(* IEC 61131-3 sources: MotionTestBenchMaster/Logical/00_AID/Libraries/Sidel_Libraries/Sidel_Obj (part 2) *)

(* ---- Shift_Obj.st ---- *)
FUNCTION_BLOCK PhotoCell_SftObj
	IF IN_ConfigPresent THEN
		VAR_GrippersNumber	:= LIMIT(1, IN_GrippersNumber, CST_RepetitiveArrayDim);
		VAR_Mask 			:= IN_MaskEn AND HMI.Mask;

		IF VAR_Mask THEN
			VAR_Signal := IN_WaitOn AND NOT IN_WaitOff;
		ELSE
			VAR_Signal := IO.DI_Input;
		END_IF

		HMI.On := VAR_Signal;

		OUT	:= HMI.On;

		IF IN_MachinePitch AND IN_Enable THEN
			VAR_ActualValveCounter	:= INT_TO_USINT(FC_ReminderShift(VAR_ActualValveCounter	+ 1, VAR_GrippersNumber, 0));

			IF IN_WritePresenceEnable THEN //v1.63
				SHIFT_Position.ContainerPresence	:= IO.DI_Input;
			END_IF//v1.63

			IF SHIFT_Position.ContainerPresence THEN//v1.63
				IF NOT SHIFT_Position.ContainerBurst	AND	NOT VAR_Mask THEN//v1.63
					IF NOT IO.DI_Input THEN
						HMI.ConsecutiveErrors	:= SEL((IN_MStopConsecutiveValue > 0), 0,HMI.ConsecutiveErrors + 1);
						HMI.AbsoluteErrors		:= SEL((IN_CBlockAbsoluteValue > 0), 0, HMI.AbsoluteErrors + 1);
						HMI.TotalErrors			:= SEL((IN_MStopAbsoluteValue > 0), HMI.TotalErrors, HMI.TotalErrors + 1);

						VAR_RepetitiveCounterArray[VAR_ActualValveCounter]	:= SEL((IN_CBlockRepetitiveValue > 0), 0, VAR_RepetitiveCounterArray[VAR_ActualValveCounter] + 1);
						SHIFT_Position.ContainerPresence	:= FALSE;//v1.63

						IF VAR_RepetitiveCounterArray[VAR_ActualValveCounter] > IN_CBlockRepetitiveValue THEN
							OUT_CBlockRepetitive	:= TRUE;
						END_IF
					ELSE
						VAR_RepetitiveCounterArray[VAR_ActualValveCounter]	:= 0;
						HMI.ConsecutiveErrors	:= 0;//v1.63
					END_IF
				ELSE//v1.63
					VAR_RepetitiveCounterArray[VAR_ActualValveCounter]	:= 0;
					HMI.ConsecutiveErrors	:= 0;
				END_IF//v1.63
			END_IF

			HMI.AlwaysTrueSteps	:= SEL(VAR_EdgeChecked, HMI.AlwaysTrueSteps + 1, 0);//v1.63

			IF IN_CBlockRepetitiveValue > 0 THEN
				HMI.RepetitiveErrors	:= 0;

				FOR VAR_GrippersNumber:= 1	TO	CST_RepetitiveArrayDim	DO
					HMI.RepetitiveErrors := MAX(HMI.RepetitiveErrors, VAR_RepetitiveCounterArray[VAR_GrippersNumber]);
				END_FOR
			END_IF
		ELSIF NOT IO.DI_Input AND IN_Enable THEN
			VAR_EdgeChecked		:= TRUE;
		END_IF

		TMR_TON_TotalCounterReset(IN := IN_ResetCounters OR HMI.CounterReset, PT := T#5s);

		IF IN_ResetCounters OR HMI.CounterReset OR VAR_Mask OR NOT IN_Enable THEN
			IF NOT VAR_CounterResetMemory THEN
				VAR_CounterResetMemory	:= TRUE;

				FOR VAR_GrippersNumber:= 1 TO CST_RepetitiveArrayDim DO
					VAR_RepetitiveCounterArray[VAR_GrippersNumber]	:= 0;
					OUT_CBlockRepetitive	:= FALSE;
				END_FOR

				HMI.AlwaysTrueSteps		:= 0;
				HMI.RepetitiveErrors	:= 0;
				HMI.ConsecutiveErrors	:= 0;
				HMI.AbsoluteErrors		:= 0;
			END_IF
		ELSE
			VAR_CounterResetMemory	:= FALSE;
		END_IF

		IF TMR_TON_TotalCounterReset.Q THEN
			IF NOT VAR_TotalCounterResetMemory THEN
				VAR_TotalCounterResetMemory := TRUE;
				HMI.TotalErrors	:= 0;
			END_IF
		ELSE
			VAR_TotalCounterResetMemory := FALSE;
		END_IF

		HMI.ConfigPresent 	:= IN_ConfigPresent;
		HMI.ConfigAlarm 	:= IN_Alarm;
		HMI.Alarm 			:= OUT_CBlockAbsolute OR OUT_MStopConsecutive OR OUT_MStopAbsolute OR OUT_AlwaysTrueError;
		HMI.Wait			:= (IN_WaitOn AND NOT HMI.On) OR (IN_WaitOff AND HMI.On);
		HMI.MaskEnable		:= IN_MaskEn;

		OUT_CBlockAbsolute		:= (HMI.AbsoluteErrors 		>= IN_CBlockAbsoluteValue)		AND (IN_CBlockAbsoluteValue		> 0);
		OUT_MStopConsecutive	:= (HMI.ConsecutiveErrors 	>= IN_MStopConsecutiveValue)	AND (IN_MStopConsecutiveValue	> 0);
		OUT_MStopAbsolute		:= (HMI.AbsoluteErrors 		>= (IN_MStopAbsoluteValue + IN_CBlockAbsoluteValue))		AND (IN_MStopAbsoluteValue		> 0);	//V4.A.A.1.6.12
		OUT_AlwaysTrueError		:= (HMI.AlwaysTrueSteps		>= CST_AlwaysTrueMaxSteps)		AND (CST_AlwaysTrueMaxSteps		> 0);
	ELSE
		OUT						:= FALSE;
		OUT_CBlockRepetitive	:= FALSE;
		OUT_CBlockAbsolute		:= FALSE;
		OUT_MStopConsecutive	:= FALSE;
		OUT_MStopAbsolute		:= FALSE;
		OUT_AlwaysTrueError		:= FALSE;
		HMI.On 					:= FALSE;
		HMI.MaskEnable			:= FALSE;
		HMI.ConfigPresent 		:= FALSE;
		HMI.ConfigAlarm 		:= FALSE;
		HMI.Alarm 				:= FALSE;
		HMI.Wait				:= FALSE;
		HMI.RepetitiveErrors	:= 0;
		HMI.ConsecutiveErrors	:= 0;
		HMI.AbsoluteErrors		:= 0;
		HMI.AlwaysTrueSteps		:= 0;
	END_IF
END_FUNCTION_BLOCK

FUNCTION_BLOCK CapPhotoCell_SftObj
	IF IN_ConfigPresent THEN
		VAR_GrippersNumber	:= LIMIT(1, IN_GrippersNumber, CST_CounterArrayDim);
		VAR_Mask 			:= IN_MaskEn AND HMI.Mask;

		IF VAR_Mask THEN
			VAR_Signal := IN_WaitOn AND NOT IN_WaitOff;
		ELSE
			VAR_Signal := IO.DI_Input;
		END_IF

		HMI.On := VAR_Signal;

		OUT	:= HMI.On;

		IF IN_MachinePitch AND IN_Enable THEN
			VAR_ActualValveCounter	:= INT_TO_USINT(FC_ReminderShift(VAR_ActualValveCounter + 1, VAR_GrippersNumber, 0));

			IF SHIFT_Position.ContainerPresence AND SHIFT_Position.ClosingReleased AND NOT VAR_Mask THEN
				HMI.AlwaysTrueSteps	:= SEL(VAR_EdgeChecked, HMI.AlwaysTrueSteps + 1, 0);
				SHIFT_Position.ContainerClosed	:= IO.DI_Input;

				IF VAR_CapsReleased < 16#FFFFFFFF THEN
					VAR_CapsReleased := VAR_CapsReleased + 1;
				ELSE
					FOR VAR_i := VAR_AbsoluteErrorN TO 1 BY -1 DO
						VAR_AbsoluteCounterArray[VAR_i] := VAR_AbsoluteCounterArray[VAR_i] - (VAR_AbsoluteCounterArray[1] - 1);
					END_FOR
					VAR_CapsReleased := VAR_AbsoluteCounterArray[VAR_AbsoluteErrorN] + 1;
				END_IF

				IF NOT IO.DI_Input THEN
					HMI.ConsecutiveErrors	:= SEL((IN_MStopConsecutiveValue > 0), 0,HMI.ConsecutiveErrors + 1);
					//HMI.AbsoluteErrors		:= SEL((IN_CBlockAbsoluteValue > 0), 0, VAR_AbsoluteErrorN);	//V4.A.A.1.6.12
					HMI.TotalErrors			:= SEL((IN_CBlockAbsoluteValue > 0) OR (IN_MStopConsecutiveValue > 0), HMI.TotalErrors, HMI.TotalErrors + 1);

					VAR_RepetitiveCounterArray[VAR_ActualValveCounter] := SEL((IN_CBlockRepetitiveValue > 0), 0, VAR_RepetitiveCounterArray[VAR_ActualValveCounter] + 1);

					IF VAR_RepetitiveCounterArray[VAR_ActualValveCounter] > IN_CBlockRepetitiveValue THEN
						OUT_CBlockRepetitive	:= TRUE;
					END_IF

					IF IN_CBlockAbsoluteValue > 0 THEN
						IF IN_CBlockAbsoluteQuantity > 0 THEN
							VAR_AbsoluteCounterArray[VAR_AbsoluteErrorN] := VAR_CapsReleased;
						ELSE
							VAR_AbsoluteCounterArray[VAR_AbsoluteErrorN] := 0;
						END_IF

						VAR_AbsoluteErrorN := VAR_AbsoluteErrorN + 1;
					ELSE
						VAR_AbsoluteCounterArray[VAR_AbsoluteErrorN] := 0;
						VAR_AbsoluteErrorN := 1;
					END_IF
				ELSE
					VAR_RepetitiveCounterArray[VAR_ActualValveCounter]	:= 0;
				END_IF
			ELSE
				HMI.ConsecutiveErrors	:= 0;
			END_IF

			IF ((VAR_CapsReleased - VAR_AbsoluteCounterArray[1]) > IN_CBlockAbsoluteQuantity) AND (IN_CBlockAbsoluteQuantity > 0) THEN
				memmove(ADR(VAR_AbsoluteCounterArray[1]), ADR(VAR_AbsoluteCounterArray[2]), SIZEOF(VAR_AbsoluteCounterArray[1]) * 49);
				VAR_AbsoluteCounterArray[50] := 0;
				VAR_AbsoluteErrorN := MAX(VAR_AbsoluteErrorN - 1, 1);
			END_IF

			IF IN_CBlockRepetitiveValue > 0 THEN
				HMI.RepetitiveErrors := 0;
				FOR VAR_GrippersNumber:= 1 TO CST_CounterArrayDim DO
					HMI.RepetitiveErrors := MAX(HMI.RepetitiveErrors, VAR_RepetitiveCounterArray[VAR_GrippersNumber]);
				END_FOR
			END_IF

			HMI.AbsoluteErrors		:= SEL((IN_CBlockAbsoluteValue > 0), 0, VAR_AbsoluteErrorN - 1);	//V4.A.A.1.6.12
		ELSIF NOT IO.DI_Input AND IN_Enable THEN
			VAR_EdgeChecked := TRUE;
		ELSIF NOT IN_Enable THEN
			SHIFT_Position.ContainerClosed	:= SHIFT_Position.ContainerPresence AND SHIFT_Position.ClosingReleased;
		END_IF

		TMR_TON_TotalCounterReset(IN := IN_ResetCounters OR HMI.CounterReset, PT := T#5s);

		IF IN_ResetCounters OR HMI.CounterReset OR VAR_Mask OR NOT IN_Enable THEN
			IF NOT VAR_CounterResetMemory THEN
				VAR_CounterResetMemory	:= TRUE;

				FOR VAR_GrippersNumber:= 1 TO CST_CounterArrayDim DO
					VAR_RepetitiveCounterArray[VAR_GrippersNumber]	:= 0;
					OUT_CBlockRepetitive	:= FALSE;
				END_FOR

				memset(ADR(VAR_AbsoluteCounterArray[1]), 0, SIZEOF(VAR_AbsoluteCounterArray));
				VAR_AbsoluteErrorN := 1;

				VAR_CapsReleased		:= 0;
				HMI.AlwaysTrueSteps		:= 0;
				HMI.RepetitiveErrors	:= 0;
				//HMI.ConsecutiveErrors	:= 0;//V1.61
				HMI.AbsoluteErrors		:= 0;
			END_IF
		ELSE
			VAR_CounterResetMemory	:= FALSE;
		END_IF
		(*V1.61 Consecutive Errorors counter reset new management*)
		IF IN_ResetCountersConsecutive OR VAR_Mask OR NOT IN_Enable THEN
			IF NOT VAR_CounterConsResetMemory THEN
				VAR_CounterConsResetMemory	:= TRUE;
				HMI.ConsecutiveErrors	:= 0;
			END_IF
		ELSE
			VAR_CounterConsResetMemory	:= FALSE;
		END_IF

		IF TMR_TON_TotalCounterReset.Q THEN
			IF NOT VAR_TotalCounterResetMemory THEN
				VAR_TotalCounterResetMemory := TRUE;
				HMI.TotalErrors	:= 0;
			END_IF
		ELSE
			VAR_TotalCounterResetMemory := FALSE;
		END_IF

		HMI.ConfigPresent 	:= IN_ConfigPresent;
		HMI.ConfigAlarm 	:= IN_Alarm;
		HMI.Alarm 			:= OUT_CBlockAbsolute OR OUT_MStopConsecutive OR OUT_AlwaysTrueError;
		HMI.Wait			:= (IN_WaitOn AND NOT HMI.On) OR (IN_WaitOff AND HMI.On);
		HMI.MaskEnable		:= IN_MaskEn;

		OUT_CBlockAbsolute		:= (HMI.AbsoluteErrors 		>= IN_CBlockAbsoluteValue)		AND (IN_CBlockAbsoluteValue		> 0);
		OUT_MStopConsecutive	:= (HMI.ConsecutiveErrors 	>= IN_MStopConsecutiveValue)	AND (IN_MStopConsecutiveValue	> 0);
		OUT_AlwaysTrueError		:= (HMI.AlwaysTrueSteps		>= CST_AlwaysTrueMaxSteps)		AND (CST_AlwaysTrueMaxSteps		> 0);
	ELSE
		OUT						:= FALSE;
		OUT_CBlockRepetitive	:= FALSE;
		OUT_CBlockAbsolute		:= FALSE;
		OUT_MStopConsecutive	:= FALSE;
		OUT_AlwaysTrueError		:= FALSE;
		HMI.On 					:= FALSE;
		HMI.MaskEnable			:= FALSE;
		HMI.ConfigPresent 		:= FALSE;
		HMI.ConfigAlarm 		:= FALSE;
		HMI.Alarm 				:= FALSE;
		HMI.Wait				:= FALSE;
		HMI.RepetitiveErrors	:= 0;
		HMI.ConsecutiveErrors	:= 0;
		HMI.AbsoluteErrors		:= 0;
		HMI.AlwaysTrueSteps		:= 0;
	END_IF
END_FUNCTION_BLOCK

FUNCTION_BLOCK CapPhotoCell_SftObj_old
	IF IN_ConfigPresent THEN
		VAR_GrippersNumber	:= LIMIT(1, IN_GrippersNumber, CST_RepetitiveArrayDim);
		VAR_Mask 			:= IN_MaskEn AND HMI.Mask;

		IF VAR_Mask THEN
			VAR_Signal := IN_WaitOn AND NOT IN_WaitOff;
		ELSE
			VAR_Signal := IO.DI_Input;
		END_IF

		HMI.On := VAR_Signal;

		OUT	:= HMI.On;

		IF IN_MachinePitch AND IN_Enable THEN
			VAR_ActualValveCounter	:= INT_TO_USINT(FC_ReminderShift(VAR_ActualValveCounter + 1, VAR_GrippersNumber, 0));

			IF SHIFT_Position.ContainerPresence AND SHIFT_Position.ClosingReleased AND NOT VAR_Mask THEN
				HMI.AlwaysTrueSteps	:= SEL(VAR_EdgeChecked, HMI.AlwaysTrueSteps + 1, 0);
				SHIFT_Position.ContainerClosed	:= IO.DI_Input;

				IF NOT IO.DI_Input THEN
					HMI.ConsecutiveErrors	:= SEL((IN_MStopConsecutiveValue > 0), 0,HMI.ConsecutiveErrors + 1);
					HMI.AbsoluteErrors		:= SEL((IN_CBlockAbsoluteValue > 0), 0, HMI.AbsoluteErrors + 1);
					HMI.TotalErrors			:= SEL((IN_MStopAbsoluteValue > 0), HMI.TotalErrors, HMI.TotalErrors + 1);

					VAR_RepetitiveCounterArray[VAR_ActualValveCounter] := SEL((IN_CBlockRepetitiveValue > 0), 0, VAR_RepetitiveCounterArray[VAR_ActualValveCounter] + 1);

					IF VAR_RepetitiveCounterArray[VAR_ActualValveCounter] > IN_CBlockRepetitiveValue THEN
						OUT_CBlockRepetitive	:= TRUE;
					END_IF
				ELSE
					VAR_RepetitiveCounterArray[VAR_ActualValveCounter]	:= 0;
				END_IF
			ELSE
				HMI.ConsecutiveErrors	:= 0;
			END_IF

			IF IN_CBlockRepetitiveValue > 0 THEN
				HMI.RepetitiveErrors := 0;
				FOR VAR_GrippersNumber:= 1 TO CST_RepetitiveArrayDim DO
					HMI.RepetitiveErrors := MAX(HMI.RepetitiveErrors, VAR_RepetitiveCounterArray[VAR_GrippersNumber]);
				END_FOR
			END_IF
		ELSIF NOT IO.DI_Input AND IN_Enable THEN
			VAR_EdgeChecked := TRUE;
		ELSIF NOT IN_Enable THEN
			SHIFT_Position.ContainerClosed	:= SHIFT_Position.ContainerPresence AND SHIFT_Position.ClosingReleased;
		END_IF

		TMR_TON_TotalCounterReset(IN := IN_ResetCounters OR HMI.CounterReset, PT := T#5s);

		IF IN_ResetCounters OR HMI.CounterReset OR VAR_Mask THEN
			IF NOT VAR_CounterResetMemory THEN
				VAR_CounterResetMemory	:= TRUE;

				FOR VAR_GrippersNumber:= 1 TO CST_RepetitiveArrayDim DO
					VAR_RepetitiveCounterArray[VAR_GrippersNumber]	:= 0;
					OUT_CBlockRepetitive	:= FALSE;
				END_FOR

				HMI.AlwaysTrueSteps		:= 0;
				HMI.RepetitiveErrors	:= 0;
				HMI.ConsecutiveErrors	:= 0;
				HMI.AbsoluteErrors		:= 0;
			END_IF
		ELSE
			VAR_CounterResetMemory	:= FALSE;
		END_IF

		IF TMR_TON_TotalCounterReset.Q THEN
			IF NOT VAR_TotalCounterResetMemory THEN
				VAR_TotalCounterResetMemory := TRUE;
				HMI.TotalErrors	:= 0;
			END_IF
		ELSE
			VAR_TotalCounterResetMemory := FALSE;
		END_IF

		HMI.ConfigPresent 	:= IN_ConfigPresent;
		HMI.ConfigAlarm 	:= IN_Alarm;
		HMI.Alarm 			:= OUT_CBlockAbsolute OR OUT_MStopConsecutive OR OUT_MStopAbsolute OR OUT_AlwaysTrueError;
		HMI.Wait			:= (IN_WaitOn AND NOT HMI.On) OR (IN_WaitOff AND HMI.On);
		HMI.MaskEnable		:= IN_MaskEn;

		OUT_CBlockAbsolute		:= (HMI.AbsoluteErrors 		>= IN_CBlockAbsoluteValue)		AND (IN_CBlockAbsoluteValue		> 0);
		OUT_MStopConsecutive	:= (HMI.ConsecutiveErrors 	>= IN_MStopConsecutiveValue)	AND (IN_MStopConsecutiveValue	> 0);
		OUT_MStopAbsolute		:= (HMI.AbsoluteErrors 		>= IN_MStopAbsoluteValue)		AND (IN_MStopAbsoluteValue		> 0);
		OUT_AlwaysTrueError		:= (HMI.AlwaysTrueSteps		>= CST_AlwaysTrueMaxSteps)		AND (CST_AlwaysTrueMaxSteps		> 0);
	ELSE
		OUT						:= FALSE;
		OUT_CBlockRepetitive	:= FALSE;
		OUT_CBlockAbsolute		:= FALSE;
		OUT_MStopConsecutive	:= FALSE;
		OUT_MStopAbsolute		:= FALSE;
		OUT_AlwaysTrueError		:= FALSE;
		HMI.On 					:= FALSE;
		HMI.MaskEnable			:= FALSE;
		HMI.ConfigPresent 		:= FALSE;
		HMI.ConfigAlarm 		:= FALSE;
		HMI.Alarm 				:= FALSE;
		HMI.Wait				:= FALSE;
		HMI.RepetitiveErrors	:= 0;
		HMI.ConsecutiveErrors	:= 0;
		HMI.AbsoluteErrors		:= 0;
		HMI.AlwaysTrueSteps		:= 0;
	END_IF
END_FUNCTION_BLOCK

FUNCTION_BLOCK Ejector_SftObj
	VAR_Mask	:= HMI.Mask AND IN_MaskEn;

	(* Local *)
	IF IN_ManEn AND NOT IN_HMIAutoForce THEN
		VAR_ManOn	:= HMI.ManOn;
		VAR_Auto	:= NOT HMI.ManOff AND NOT HMI.ManOn;
	ELSE
		VAR_ManOn	:= FALSE;
		VAR_Auto	:= TRUE;
		HMI.ManOn	:= FALSE;
		HMI.ManOff	:= FALSE;
	END_IF

	IF IN_MachinePitch THEN
		VAR_AutoCnd := IN_ShiftPosition.ContainerPresence		AND (IN_ShiftPosition.ContainerBurst	OR
						(NOT IN_ShiftPosition.ContainerFilled	AND IN_FillingErrorEject) OR IN_ShiftPosition.EjectContainer) AND NOT VAR_Mask; (*V1.61*)
		IF VAR_AutoCnd AND NOT IN_SamplingModeActive THEN (*V1.61*)
			HMI.ConsecutiveErrors	:= HMI.ConsecutiveErrors	+ 1;
			HMI.AbsoluteErrors		:= HMI.AbsoluteErrors		+ 1;
			HMI.TotalErrors			:= HMI.TotalErrors			+ 1;
		ELSE
			HMI.ConsecutiveErrors	:= 0;
		END_IF(*V1.61*)

		IF IN_SamplingModeActive AND VAR_AutoCnd THEN (*V1.61*)
			IN_ShiftPosition.ContainerEjected := TRUE;(*V1.61*)
		ELSE
			IN_ShiftPosition.ContainerEjected := FALSE;(*V1.61*)
		END_IF
	END_IF

	TMR_TON_TotalCounterReset(IN := IN_ResetCounters OR HMI.CounterReset, PT := T#5s);

	IF IN_ResetCounters OR HMI.CounterReset THEN
		IF NOT VAR_CounterResetMemory THEN
			VAR_CounterResetMemory	:= TRUE;
			HMI.ConsecutiveErrors	:= 0;
			HMI.AbsoluteErrors		:= 0;
		END_IF
	ELSE
		VAR_CounterResetMemory	:= FALSE;
	END_IF

	IF TMR_TON_TotalCounterReset.Q THEN
		IF NOT VAR_TotalCounterResetMemory THEN
			VAR_TotalCounterResetMemory := TRUE;
			HMI.TotalErrors	:= 0;
		END_IF
	ELSE
		VAR_TotalCounterResetMemory := FALSE;
	END_IF

	IF IN_ConfigPresent THEN
		IF IN_Enable THEN
			IF VAR_Auto THEN
				VAR_ValveOpened := VAR_AutoCnd;
			ELSIF VAR_ManOn THEN
				VAR_ValveOpened := TRUE;
			ELSE
				VAR_ValveOpened := FALSE;
			END_IF
		ELSIF NOT IN_ConfigType THEN
			VAR_ValveOpened := FALSE;
		END_IF
		VAR_ValveClosed := NOT VAR_ValveOpened;

		OUT						:= VAR_ValveOpened;
		OUT_CBlockAbsolute		:= (HMI.AbsoluteErrors 		>= IN_CBlockAbsoluteValue)		AND (IN_CBlockAbsoluteValue		> 0);
		OUT_MStopConsecutive	:= (HMI.ConsecutiveErrors 	>= IN_MStopConsecutiveValue)	AND (IN_MStopConsecutiveValue	> 0);
	ELSE
		VAR_ValveOpened			:= FALSE;
		VAR_ValveClosed			:= FALSE;
		OUT						:= FALSE;
		OUT_CBlockAbsolute		:= 0;
		OUT_MStopConsecutive	:= 0;
	END_IF

	(* HMI *)
	HMI.ManEnable		:= IN_ManEn;
	HMI.ConfigPresent	:= IN_ConfigPresent;
	HMI.MaskEnable		:= IN_MaskEn;
	HMI.Alarm 			:= OUT_CBlockAbsolute OR OUT_MStopConsecutive;

	(* IO *)
	IO.DO_Opened	:= VAR_ValveOpened;
	IO.DO_Closed	:= VAR_ValveClosed;
	HMI.Out			:= IO.DO_Opened;
END_FUNCTION_BLOCK

(* ---- Sidel_Obj.fun ---- *)
FUNCTION_BLOCK Analog_In_Direct_Inverse
	VAR_INPUT
		IN_ConfigPresent : BOOL;
		IN_Simulation : BOOL;
		IN_0_20mA : BOOL;
		IN_FaultOutMode : USINT; (*LowOnFault(1) ; HighOnFault (2) HoldOnFault (0)*)
		IN_EngScale : BOOL;
		IN_CompareMode : USINT; (*0 = Off, 1 = PV_Greater_SP, 2 = PV_Less_SP, 3 = PV_Equal_SP, 4 = On*)
		IN_ScaleLOW : REAL;
		IN_ScaleHIGH : REAL;
		IN_AlarmEn : BOOL;
		IN_MaskEn : BOOL;
		IN_ConfigPopup : BOOL;
		IN_Reset : BOOL; (*Reset Analog Channel Alarm*)
		IN_ActualSP : REAL; (*Signal Input Actual Set Point*)
		IN_MinDev : REAL; (*To Set Point Low Deviation (for SP obtained)*)
		IN_MaxDev : REAL; (*To Set Point High Deviation (for SP obtained)*)
		IN_WaitDelay : TIME;
		IN_HighLimitEn : BOOL;
		IN_HighLimitSP : REAL;
		IN_HighLimitHyst : REAL;
		IN_HighLimitDelay : TIME;
		IN_LowLimitEn : BOOL;
		IN_LowLimitSP : REAL;
		IN_LowLimitHyst : REAL;
		IN_LowLimitDelay : TIME;
		IN_Direct_Inverse : BOOL; (*Read Mode: "0" for Direct "1" for Inverse*)
		IN_Delta : REAL; (*Delta Value for Real Component Height*)
	END_VAR
	VAR_OUTPUT
		OUT_ActValue : REAL; (*Manipulated value*)
		OUT_SpReached : BOOL; (*Output Set Point Reached*)
		OUT_HighLimit : BOOL;
		OUT_LowLimit : BOOL;
		OUT_Alarm : BOOL; (*Output Fault*)
		OUT_RawOverflow : BOOL; (*Output Fault*)
		OUT_RawUnderflow : BOOL; (*Output Fault*)
	END_VAR
	VAR_IN_OUT
		IO : IO_Analog_IN_Type;
		HMI : HMI_Analog_IN_Type;
	END_VAR
	VAR
		VAR_Fault : BOOL; (*Alarm Output for Fault or Warning*)
		VAR_Mask : BOOL;
		VAR_Out : REAL;
		VAR_ChannelActive : BOOL;
		VAR_Wait : BOOL;
		VAR_iFault : BOOL;
		VAR_SpReached : BOOL;
		LCRLimScal_0_20mA : LCRLimScal;
		LCRLimScal_4_20mA : LCRLimScal;
		TMR_TON_HighLimitDelay : TON;
		TMR_TON_LowLimitDelay : TON;
		TMR_TOF_SpReached : TOF;
	END_VAR
END_FUNCTION_BLOCK

FUNCTION_BLOCK Analog_In
	VAR_INPUT
		IN_ConfigPresent : BOOL;
		IN_Simulation : BOOL;
		IN_0_20mA : BOOL;
		IN_FaultOutMode : USINT; (*LowOnFault(1) ; HighOnFault (2) HoldOnFault (0)*)
		IN_EngScale : BOOL;
		IN_CompareMode : USINT; (*0 = Off, 1 = PV_Less_SP, 2 = PV_Greater_SP, 3 = PV_Equal_SP, 4 = Reached On*)
		IN_ScaleLOW : REAL;
		IN_ScaleHIGH : REAL;
		IN_AlarmEn : BOOL;
		IN_MaskEn : BOOL;
		IN_ConfigPopup : BOOL;
		IN_Reset : BOOL; (*Reset Analog Channel Alarm*)
		IN_ActualSP : REAL; (*Signal Input Actual Set Point*)
		IN_MinDev : REAL; (*To Set Point Low Deviation (for SP obtained)*)
		IN_MaxDev : REAL; (*To Set Point High Deviation (for SP obtained)*)
		IN_WaitDelay : TIME;
		IN_HighLimitEn : BOOL;
		IN_HighLimitSP : REAL;
		IN_HighLimitHyst : REAL;
		IN_HighLimitDelay : TIME;
		IN_LowLimitEn : BOOL;
		IN_LowLimitSP : REAL;
		IN_LowLimitHyst : REAL;
		IN_LowLimitDelay : TIME;
		IN_TotPulseWeight : REAL;
		IN_TotType : USINT;
		IN_PLCCounterEn : BOOL;
		IN_PLCCounterSP : REAL;
		IN_PLCCounterReset : BOOL;
		IN_HMITotEn : BOOL;
		IN_HMITotReset : BOOL;
	END_VAR
	VAR_OUTPUT
		OUT_ActValue : REAL; (*Manipulated value*)
		OUT_SpReached : BOOL; (*Output Set Point Reached*)
		OUT_HighLimit : BOOL;
		OUT_LowLimit : BOOL;
		OUT_Alarm : BOOL; (*Output Fault*)
		OUT_RawOverflow : BOOL; (*Output Fault*)
		OUT_RawUnderflow : BOOL; (*Output Fault*)
		OUT_PLCCounterReached : BOOL; (*Output Fault*)
	END_VAR
	VAR_IN_OUT
		IO : IO_Analog_IN_Type;
		HMI : HMI_Analog_IN_Type;
	END_VAR
	VAR
		VAR_Fault : BOOL; (*Alarm Output for Fault or Warning*)
		VAR_Mask : BOOL;
		VAR_Out : REAL;
		VAR_ChannelActive : BOOL;
		VAR_Wait : BOOL;
		VAR_iFault : BOOL;
		VAR_SpReached : BOOL;
		LCRLimScal_0_20mA : LCRLimScal;
		LCRLimScal_4_20mA : LCRLimScal;
		HMITotalizer : AnalogTotalizer;
		PLCCounter : AnalogTotalizer;
		TMR_TON_HighLimitDelay : TON;
		TMR_TON_LowLimitDelay : TON;
		TMR_TOF_SpReached : TOF;
		TON_ChannelOk : TON;
	END_VAR
END_FUNCTION_BLOCK

FUNCTION_BLOCK GateDoorDigital_Obj
	VAR_INPUT
		IN_ConfigPresent : BOOL; (*Configuration: Device Present*)
		IN_Alarm : BOOL; (*Configuration: Timeout Alarm Control Enable*)
		IN_AlarmOpenReq : BOOL; (*Control: On State Time Out Alarm Request*)
		IN_AlarmCloseReq : BOOL; (*Control: Off State Time Out Alarm Request*)
		IN_SwitchDelay : TIME; (*Time: Row Input Switching State Display Delay*)
		IN_WaitOpen : BOOL; (*Control: On State Wait Request*)
		IN_WaitClose : BOOL; (*Control: Off State Wait Request*)
		IN_OnDelay : TIME; (*Time: State On / Alarm On Time Delay*)
		IN_OffDelay : TIME; (*Time: State Off / Alarm Off Time Delay*)
		IN_Reset : BOOL; (*Control: Alarm Reset Push Button*)
		IN_SafetyClosed : BOOL; (*From Safety: Gate Closed*)
		IN_SafetyShortCircuit : BOOL; (*From Safety: Short circuit or 1oo2*)
	END_VAR
	VAR_OUTPUT
		OUT_Opened : BOOL; (*OUT: Gate Opened*)
		OUT_Closed : BOOL; (*OUT: Gate Closed*)
		OUT_Alarm : BOOL; (*State On / Off Time Out Alarm*)
	END_VAR
	VAR_IN_OUT
		IO_Production : IO_Digital_IN_Type; (*State: Digital Input Structure*)
		HMI : HMI_GateDoor_Type;
	END_VAR
	VAR
		TMR_TON_ProdSwOn : TON;
		TMR_TON_ProdSwOff : TON;
		TMR_TON_CleanSwOn : TON;
		TMR_TON_CleanSwOff : TON;
		TMR_TON_ProdOnAlarm : TON;
		TMR_TON_ProdOffAlarm : TON;
		TMR_TON_CleanOnAlarm : TON;
		TMR_TON_CleanOffAlarm : TON;
		VAR_Signal : BOOL;
		VAR_ProdFault : BOOL;
		VAR_CleanFault : BOOL;
	END_VAR
END_FUNCTION_BLOCK

FUNCTION_BLOCK Analog_In_Multiscale
	VAR_INPUT
		IN_ConfigPresent : BOOL;
		IN_Simulation : BOOL;
		IN_0_20mA : BOOL;
		IN_MaskEn : BOOL;
		IN_Reset : BOOL; (*Reset Analog Channel Alarm*)
		IN_FaultOutMode : USINT; (*LowOnFault(1) ; HighOnFault (2) HoldOnFault (0)*)
		IN_EngScale : BOOL;
		IN_AlarmEn : BOOL;
		IN_ConfigPopup : BOOL;
		IN_PLCCounterEn : BOOL;
		IN_CompareMode : USINT; (*0 = Off, 1 = PV_Greater_SP, 2 = PV_Less_SP, 3 = PV_Equal_SP, 4 = On*)
		IN_ScaleIndex : USINT; (*0..3 = Array Requested*)
		IN_Scale : ARRAY[0..3] OF IN_Analog_Multiscale; (*0..3 = Arrays for Different Scale*)
	END_VAR
	VAR_OUTPUT
		OUT_Alarm : BOOL; (*Output Fault*)
		OUT_SpReached : BOOL; (*Output Set Point Reached*)
		OUT_RawOverflow : BOOL; (*Output Analog Fault*)
		OUT_RawUnderflow : BOOL; (*Output Analog Fault*)
		OUT_Scale : ARRAY[0..3] OF OUT_Analog_Multiscale;
	END_VAR
	VAR_IN_OUT
		IO : IO_Analog_IN_Type;
		HMI : HMI_Analog_Multiscale_Type;
	END_VAR
	VAR
		VAR_Fault : BOOL; (*Alarm Output for Fault or Warning*)
		VAR_Mask : BOOL;
		VAR_ChannelActive : BOOL;
		VAR_Wait : BOOL;
		VAR_iFault : BOOL;
		VAR_SpReached : BOOL;
		VAR_Index : USINT;
		VAR_Out : REAL;
		LCRLimScal_0_20mA : LCRLimScal;
		LCRLimScal_4_20mA : LCRLimScal;
		HMITotalizer : AnalogTotalizer;
		PLCCounter : AnalogTotalizer;
		TMR_TON_HighLimitDelay : TON;
		TMR_TON_LowLimitDelay : TON;
		TMR_TOF_SpReached : TOF;
	END_VAR
END_FUNCTION_BLOCK

FUNCTION_BLOCK Analog_In_Multicompare
	VAR_INPUT
		IN_ConfigPresent : BOOL;
		IN_Simulation : BOOL;
		IN_0_20mA : BOOL;
		IN_MaskEn : BOOL;
		IN_Reset : BOOL; (*Reset Analog Channel Alarm*)
		IN_FaultOutMode : USINT; (*LowOnFault(1) ; HighOnFault (2) HoldOnFault (0)*)
		IN_EngScale : BOOL;
		IN_AlarmEn : BOOL;
		IN_ConfigPopup : BOOL;
		IN_PLCCounterEn : BOOL;
		IN_CompareMode : USINT; (*0 = Off, 1 = PV_Greater_SP, 2 = PV_Less_SP, 3 = PV_Equal_SP, 4 = On*)
		IN_ScaleIndex : USINT; (*0..3 = Array Requested*)
		IN_Scale : ARRAY[0..3] OF IN_Analog_Multiscale; (*0..3 = Arrays for Different Scale*)
	END_VAR
	VAR_OUTPUT
		OUT_Alarm : BOOL; (*Output Fault*)
		OUT_SpReached : BOOL; (*Output Set Point Reached*)
		OUT_RawOverflow : BOOL; (*Output Analog Fault*)
		OUT_RawUnderflow : BOOL; (*Output Analog Fault*)
		OUT_Scale : ARRAY[0..3] OF OUT_Analog_Multiscale;
	END_VAR
	VAR_IN_OUT
		IO : IO_Analog_IN_Type;
		HMI : HMI_Analog_Multiscale_Type;
	END_VAR
	VAR
		VAR_Fault : BOOL; (*Alarm Output for Fault or Warning*)
		VAR_Mask : BOOL;
		VAR_ChannelActive : BOOL;
		VAR_Wait : BOOL;
		VAR_iFault : BOOL;
		VAR_SpReached : BOOL;
		VAR_Index : USINT;
		VAR_Out : REAL;
		LCRLimScal_0_20mA : LCRLimScal;
		LCRLimScal_4_20mA : LCRLimScal;
		HMITotalizer : AnalogTotalizer;
		PLCCounter : AnalogTotalizer;
		TMR_TON_HighLimitDelay : TON;
		TMR_TON_LowLimitDelay : TON;
		TMR_TOF_SpReached : TOF;
	END_VAR
END_FUNCTION_BLOCK

FUNCTION_BLOCK Digital_Obj
	VAR_INPUT
		IN_ConfigPresent : BOOL; (*Configuration: Device Present*)
		IN_Alarm : BOOL; (*Configuration: Timeout Alarm Control Enable*)
		IN_AlarmOnReq : BOOL; (*Control: On State Time Out Alarm Request*)
		IN_AlarmOffReq : BOOL; (*Control: Off State Time Out Alarm Request*)
		IN_SwitchDelay : TIME; (*Time: Row Input Switching State Display Delay*)
		IN_WaitOn : BOOL; (*Control: On State Wait Request*)
		IN_WaitOff : BOOL; (*Control: Off State Wait Request*)
		IN_OnDelay : TIME; (*Time: State On / Alarm On Time Delay*)
		IN_OffDelay : TIME; (*Time: State Off / Alarm Off Time Delay*)
		IN_Reset : BOOL; (*Control: Alarm Reset Push Button*)
		IN_MaskEn : BOOL; (*Control: Mask Enable*)
	END_VAR
	VAR_OUTPUT
		OUT : BOOL; (*State Switching Delayed*)
		OUT_OnDelayed : BOOL; (*State On Time Delayed*)
		OUT_OffDelayed : BOOL; (*State Off Time Delayed*)
		OUT_Alarm : BOOL; (*State On / Off Time Out Alarm*)
	END_VAR
	VAR_IN_OUT
		IO : IO_Digital_IN_Type; (*State: Digital Input Structure*)
		HMI : HMI_DI_Type;
	END_VAR
	VAR
		TMR_TON_SwOn : TON;
		TMR_TON_SwOff : TON;
		TMR_TON_OnTime : TON;
		TMR_TON_OffTime : TON;
		TMR_TON_OnAlarm : TON;
		TMR_TON_OffAlarm : TON;
		VAR_Signal : BOOL;
		VAR_Mask : BOOL;
	END_VAR
END_FUNCTION_BLOCK

FUNCTION_BLOCK Motor_Std_Fw_Bw
	VAR_INPUT
		IN_ConfigPresent : BOOL;
		IN_Simulation : BOOL;
		IN_Enable : BOOL; (*Safety OK ( True if not used)*)
		IN_AutoCnd : BOOL; (*Automation Logic Input*)
		IN_Backward : BOOL; (*Direction Reverse*)
		IN_Reset : BOOL; (*Fault Reset*)
		IN_HMIAutoForce : BOOL;
		IN_FbkCheck : BOOL;
		IN_ManEn : BOOL;
		IN_MaskEn : BOOL;
		IN_FBKDelay : TIME := T#500ms; (*Time: Running Control Delay*)
		IN_ConfigType : BOOL; (*Configuration: Type TRUE = Phoenix FALSE = Contactor*)
	END_VAR
	VAR_OUTPUT
		OUT_Running : BOOL; (*Motor On*)
		OUT_ContactorFBKFault : BOOL;
		OUT_OverloadFault : BOOL;
		OUT_Alarm : BOOL; (*Output for Alarm*)
		OUT_IsolatedFault : BOOL;
	END_VAR
	VAR_IN_OUT
		IO : IO_Motor_FwBw_Type;
		HMI : HMI_Motor_Type;
	END_VAR
	VAR
		TMR_TOF : TON;
		TMR_TON : TON;
		VAR_ContactorFBK : BOOL;
		VAR_DiFault : BOOL;
		VAR_Overload : BOOL;
		VAR_Mask : BOOL;
		VAR_Auto : BOOL;
		VAR_Fault : BOOL; (*Alarm Output for Fault or Warning*)
		VAR_FirstCycle : BOOL;
		VAR_Isolated : BOOL;
		zzEdge00000 : BOOL;
	END_VAR
END_FUNCTION_BLOCK

FUNCTION_BLOCK Motor_Std
	VAR_INPUT
		IN_ConfigPresent : BOOL;
		IN_Simulation : BOOL;
		IN_Enable : BOOL; (*Safety OK ( True if not used)*)
		IN_AutoCnd : BOOL; (*Automation Logic Input*)
		IN_Reset : BOOL; (*Fault Reset*)
		IN_HMIAutoForce : BOOL;
		IN_ManEn : BOOL;
		IN_MaskEn : BOOL;
		IN_FBKDelay : TIME := T#500ms; (*Time: Running Control Delay*)
		IN_ConfigType : BOOL; (*Configuration: Type TRUE = Phoenix FALSE = Contactor*)
	END_VAR
	VAR_OUTPUT
		OUT_Running : BOOL; (*Motor On*)
		OUT_IsolatedFault : BOOL;
		OUT_ContactorFBKFault : BOOL;
		OUT_OverloadFault : BOOL;
		OUT_Alarm : BOOL; (*Output for Alarm*)
	END_VAR
	VAR_IN_OUT
		IO : IO_Motor_Type;
		HMI : HMI_Motor_Type;
	END_VAR
	VAR
		TMR_TOF : TON;
		TMR_TON : TON;
		VAR_ContactorFBK : BOOL;
		VAR_Isolated : BOOL;
		VAR_Overload : BOOL;
		VAR_Mask : BOOL;
		VAR_Auto : BOOL;
		VAR_Fault : BOOL; (*Alarm Output for Fault or Warning*)
		VAR_FirstCycle : BOOL;
		zzEdge00000 : BOOL;
	END_VAR
END_FUNCTION_BLOCK

FUNCTION_BLOCK UVtronic_Std
	VAR_INPUT
		IN_ConfigPresent : BOOL;
		IN_Simulation : BOOL;
		IN_Enable : BOOL; (*Safety OK ( True if not used)*)
		IN_AutoCnd : BOOL; (*Automation Logic Input*)
		IN_Reset : BOOL; (*Fault Reset*)
		IN_HMIAutoForce : BOOL;
		IN_ManEn : BOOL;
		IN_MaskEn : BOOL;
		IN_FBKDelay : TIME := T#500ms; (*Time: Running Control Delay*)
		IN_ConfigType : BOOL; (*Configuration: Type TRUE = Phoenix FALSE = Contactor*)
	END_VAR
	VAR_OUTPUT
		OUT_Running : BOOL; (*Motor On*)
		OUT_NotReady : BOOL;
		OUT_GeneralFault : BOOL;
		OUT_ContactorFBKFault : BOOL;
		OUT_OverloadFault : BOOL;
		OUT_Alarm : BOOL; (*Output for Alarm*)
	END_VAR
	VAR_IN_OUT
		IO : IO_UVtronic_Type;
		HMI : HMI_Motor_Type;
	END_VAR
	VAR
		TMR_TOF : TON;
		TMR_TON : TON;
		VAR_ContactorFBK : BOOL;
		VAR_NotReady : BOOL;
		VAR_GeneralFault : BOOL;
		VAR_Overload : BOOL;
		VAR_Mask : BOOL;
		VAR_Auto : BOOL;
		VAR_Fault : BOOL; (*Alarm Output for Fault or Warning*)
		VAR_FirstCycle : BOOL;
		zzEdge00000 : BOOL;
	END_VAR
END_FUNCTION_BLOCK

FUNCTION_BLOCK Motor_FC280_Vfd
	VAR_INPUT
		IN_Simulation : BOOL;
		IN_ConfigPresent : BOOL; (*Configuration: Device Present*)
		IN_Enable : BOOL;
		IN_AutoCnd : BOOL; (*Automation Logic Input*)
		IN_AutoSpeed : REAL;
		IN_Reverse : BOOL;
		IN_FrequencyMin : REAL;
		IN_FrequencyMax : REAL;
		IN_ManEn : BOOL; (*Control: Manual On Enabled*)
		IN_MaskEn : BOOL; (*Control: Alarm Mask Enable*)
		IN_Reset : BOOL; (*Control: Alarm Reset Push Button*)
		IN_HMIAutoForce : BOOL;
		IN_QuickStopCmd : BOOL; (*Control: Quick Stop Command (TRUE = Quick Stop)*)
		IN_JOGMode : BOOL; (*Control: JOG Mode (if TRUE)*)
		IN_JOGCnd : BOOL; (*Control: JOG Running Condition*)
		IN_CoastingCmd : BOOL; (*Control: Coasting (TRUE = Coasting)*)
		IN_FCD : BOOL; (*Configuration: Drive Type FCD V4.A.A.1.6.13*)
		IN_FBKDelay : TIME := T#500ms; (*Time: Running Control Delay*)
		IN_SafetyCtrlEn : BOOL; (*Configuration: Drive SafeOFF Enabled TRUE = Control Enabled*)
		IN_ScaleMax : REAL := 100.0; (*Configuration: Drive speed Scale Maximum Value*)
	END_VAR
	VAR_OUTPUT
		OUT_InOperation : BOOL;
		OUT_DriveSafetyFBKFault : BOOL; (*Safety XOR 37*)
		OUT_DriveFault : BOOL; (*Drive fault (from STW) or high current*)
		OUT_IsolatedFault : BOOL;
		OUT_OverloadFault : BOOL;
		OUT_ActualSpeed : REAL;
		OUT_ActualFrequency : REAL;
		OUT_ActualCurrent : REAL;
		OUT_ActualTorque : REAL;
		OUT_ActualPower : REAL;
		OUT_ActualSpeedRPM : REAL;
		OUT_Warning : BOOL; (*Drive warning (from STW)*)
		OUT_SpeedReferece : BOOL;
	END_VAR
	VAR_IN_OUT
		HMI_Danfoss : HMI_Danfoss_Diag_Type;
		HMI_Motor : HMI_Motor_FC_Type;
		IO_DanfossFC280 : IO_PLK_DanfossFC280_Drive_Type;
		IO_MotorFC280 : IO_MotorFC280_Type;
	END_VAR
	VAR
		VAR_RecSTW : Danfoss_STW_Type;
		VAR_RecDI : Danfoss_DI_Type; (*V4.A.A.1.6.13*)
		VAR_SendCTW : Danfoss_CTW_Type;
		TMR_TON_CurrentHigh : TON;
		TMR_TON_FaultFilter : TON;
		TMR_TON_FBKTimeOut : TON;
		TMR_TON_RFeedBack : TON;
		TMR_TON_WarningFilter : TON;
		VAR_CurrentHigh : BOOL;
		VAR_Event : Danfoss_Event_Type;
		VAR_Fault : BOOL; (*Memory Output Generic*)
		VAR_FirstCycle : BOOL;
		VAR_AutoSpeed : REAL;
		VAR_Isolated : BOOL;
		VAR_Overload : BOOL;
		VAR_Auto : BOOL;
		VAR_Mask : BOOL;
		VAR_Start : BOOL; (*Motor start*)
		zzEdge00000 : BOOL;
		zzEdge1 : BOOL;
		zzEdge2 : BOOL;
		zzEdge3 : BOOL;
		zzEdge4 : BOOL;
		zzEdge5 : BOOL;
	END_VAR
END_FUNCTION_BLOCK

FUNCTION_BLOCK Motor_Vfd
	VAR_INPUT
		IN_Simulation : BOOL;
		IN_ConfigPresent : BOOL; (*Configuration: Device Present*)
		IN_Enable : BOOL;
		IN_AutoCnd : BOOL; (*Automation Logic Input*)
		IN_AutoSpeed : REAL;
		IN_Reverse : BOOL;
		IN_FrequencyMin : REAL;
		IN_FrequencyMax : REAL;
		IN_ManEn : BOOL; (*Control: Manual On Enabled*)
		IN_MaskEn : BOOL; (*Control: Alarm Mask Enable*)
		IN_Reset : BOOL; (*Control: Alarm Reset Push Button*)
		IN_HMIAutoForce : BOOL;
		IN_QuickStopCmd : BOOL; (*Control: Quick Stop Command (TRUE = Quick Stop)*)
		IN_JOGMode : BOOL; (*Control: JOG Mode (if TRUE)*)
		IN_JOGCnd : BOOL; (*Control: JOG Running Condition*)
		IN_CoastingCmd : BOOL; (*Control: Coasting (TRUE = Coasting)*)
		IN_FCD : BOOL; (*Configuration: Drive Type FCD V4.A.A.1.6.13*)
		IN_FBKDelay : TIME := T#500ms; (*Time: Running Control Delay*)
		IN_SafetyCtrlEn : BOOL; (*Configuration: Drive SafeOFF Enabled TRUE = Control Enabled*)
		IN_ScaleMax : REAL := 100.0; (*Configuration: Drive speed Scale Maximum Value*)
	END_VAR
	VAR_OUTPUT
		OUT_InOperation : BOOL;
		OUT_DriveSafetyFBKFault : BOOL; (*Safety XOR 37*)
		OUT_DriveFault : BOOL; (*Drive fault (from STW) or high current*)
		OUT_IsolatedFault : BOOL;
		OUT_OverloadFault : BOOL;
		OUT_ActualSpeed : REAL;
		OUT_ActualFrequency : REAL;
		OUT_ActualCurrent : REAL;
		OUT_ActualTorque : REAL;
		OUT_ActualPower : REAL;
		OUT_ActualSpeedRPM : REAL;
		OUT_Warning : BOOL; (*Drive warning (from STW)*)
		OUT_SpeedReferece : BOOL;
		OUT_ActualDigitalState : Danfoss_DI_Type; (*V1.7.2*)
	END_VAR
	VAR_IN_OUT
		HMI_Danfoss : HMI_Danfoss_Diag_Type;
		HMI_Motor : HMI_Motor_FC_Type;
		IO_Danfoss : IO_PLK_Danfoss_Drive_Type;
		IO_Motor : IO_Motor_Type;
	END_VAR
	VAR
		VAR_RecSTW : Danfoss_STW_Type;
		VAR_RecDI : Danfoss_DI_Type; (*V4.A.A.1.6.13*)
		VAR_SendCTW : Danfoss_CTW_Type;
		TMR_TON_CurrentHigh : TON;
		TMR_TON_FaultFilter : TON;
		TMR_TON_FBKTimeOut : TON;
		TMR_TON_RFeedBack : TON;
		TMR_TON_WarningFilter : TON;
		VAR_CurrentHigh : BOOL;
		VAR_Event : Danfoss_Event_Type;
		VAR_Fault : BOOL; (*Memory Output Generic*)
		VAR_FirstCycle : BOOL;
		VAR_AutoSpeed : REAL;
		VAR_Isolated : BOOL;
		VAR_Overload : BOOL;
		VAR_Auto : BOOL;
		VAR_Mask : BOOL;
		VAR_Start : BOOL; (*Motor start*)
		zzEdge00000 : BOOL;
	END_VAR
END_FUNCTION_BLOCK

FUNCTION_BLOCK Valve_Dig_Mac (*Valve Control: Digital*)
	VAR_INPUT
		IN_ConfigPresent : BOOL; (*Configuration: Device Present*)
		IN_ConfigType : BOOL; (*Configuration: Device Type (0: Monostable - 1: Bistable)*)
		IN_Simulation : BOOL;
		IN_ConfigPositionSensorOpened : BOOL;
		IN_ConfigPositionSensorClosed : BOOL;
		IN_StrokeTime : TIME;
		IN_Enable : BOOL;
		IN_AutoCnd : BOOL; (*Automation Logic Input*)
		IN_EnableCnd : BOOL;
		IN_Cnd : BOOL;
		IN_FlipEnable : BOOL;
		IN_FlipRequest : BOOL;
		IN_FlipTime : TIME;
		IN_Reset : BOOL; (*Fault Reset*)
		IN_HMIAutoForce : BOOL;
		IN_ManEn : BOOL;
		IN_MaskEn : BOOL;
	END_VAR
	VAR_OUTPUT
		OUT : BOOL; (*Stroke done*)
		OUT_Alarm : BOOL; (*Fault Output for Alarm*)
		OUT_OpenedFiltered : BOOL; (*Stroke done*)
		OUT_ClosedFiltered : BOOL; (*Stroke done*)
		OUT_FlipDone : BOOL;
	END_VAR
	VAR_IN_OUT
		IO : IO_ValveMac_Type;
		HMI : HMI_Valve_Type;
	END_VAR
	VAR
		VAR_Enable : BOOL;
		VAR_iFault : BOOL;
		VAR_Mask : BOOL;
		TMR_TOF_FeedBackOpen : TOF;
		TMR_TOF_FeedBackClose : TOF;
		VAR_ManOn : BOOL;
		VAR_Auto : BOOL;
		MAX_Flip_Time : TIME := T#1S;
		VAR_AutoCnd : BOOL;
		VAR_ConfigPosition : BOOL;
		TMR_TON_ControlEnableDelay : TON;
		TMR_TON_Opened : TON;
		TMR_TON_Closed : TON;
		VAR_FeedBackOpen : BOOL;
		VAR_FeedBackClose : BOOL;
		VAR_ValveOpened : BOOL;
		VAR_Fault : BOOL;
		TMR_TP_Block : TP_Reset;
		TMR_TP_Release : TP_Reset;
		TMR_TON_Flip : TON;
		VAR_ValveClosed : BOOL;
		TMR_TON_ClosedFilter : TON;
		TMR_TON_OpenedFilter : TON;
	END_VAR
END_FUNCTION_BLOCK

FUNCTION_BLOCK Valve_Dig (*Valve Control: Digital*)
	VAR_INPUT
		IN_ConfigPresent : BOOL; (*Configuration: Device Present*)
		IN_ConfigType : BOOL; (*Configuration: Device Type (0: Monostable - 1: Bistable)*)
		IN_ConfigNormallyOpen : BOOL; (*Configuration: Device Type (0: Normally Closed - 1: Normally Open) v1.5*)
		IN_Simulation : BOOL;
		IN_ConfigPositionSensorOpened : BOOL;
		IN_ConfigPositionSensorClosed : BOOL;
		IN_StrokeTime : TIME;
		IN_Enable : BOOL;
		IN_AutoCnd : BOOL; (*Automation Logic Input*)
		IN_EnableCnd : BOOL;
		IN_Cnd : BOOL;
		IN_FlipEnable : BOOL;
		IN_FlipRequest : BOOL;
		IN_FlipTime : TIME;
		IN_Reset : BOOL; (*Fault Reset*)
		IN_HMIAutoForce : BOOL;
		IN_ManEn : BOOL;
		IN_MaskEn : BOOL;
	END_VAR
	VAR_OUTPUT
		OUT : BOOL; (*Stroke done*)
		OUT_Alarm : BOOL; (*Fault Output for Alarm*)
		OUT_OpenedFiltered : BOOL; (*Stroke done*)
		OUT_ClosedFiltered : BOOL; (*Stroke done*)
		OUT_FlipDone : BOOL;
	END_VAR
	VAR_IN_OUT
		IO : IO_Valve_Type;
		HMI : HMI_Valve_Type;
	END_VAR
	VAR
		VAR_Enable : BOOL;
		VAR_iFault : BOOL;
		VAR_Mask : BOOL;
		TMR_TOF_FeedBackOpen : TOF;
		TMR_TOF_FeedBackClose : TOF;
		VAR_ManOn : BOOL;
		VAR_Auto : BOOL;
		MAX_Flip_Time : TIME := T#1S;
		VAR_AutoCnd : BOOL;
		VAR_ConfigPosition : BOOL;
		TMR_TON_ControlEnableDelay : TON;
		TMR_TON_Opened : TON;
		TMR_TON_Closed : TON;
		VAR_FeedBackOpen : BOOL;
		VAR_FeedBackClose : BOOL;
		VAR_ValveOpened : BOOL;
		VAR_Fault : BOOL;
		TMR_TON_Flip : TON;
		VAR_ValveClosed : BOOL;
		TMR_TON_ClosedFilter : TON;
		TMR_TON_OpenedFilter : TON;
	END_VAR
END_FUNCTION_BLOCK

FUNCTION_BLOCK Valve_Mod
	VAR_INPUT
		IN_ConfigPresent : BOOL;
		IN_Simulation : BOOL;
		IN_ConfigPositionSensorOpened : BOOL;
		IN_ConfigPositionSensorClosed : BOOL;
		IN_ConfigPositionAnalogFBK : BOOL;
		IN_StrokeTime : TIME;
		IN_ConfigNormallyOpen : BOOL;
		IN_Enable : BOOL;
		IN_AutoCnd : BOOL;
		IN_AutoVal : REAL;
		IN_OpeningRampEn : BOOL;
		IN_OpeningRampValue : REAL;
		IN_ClosingRampEn : BOOL;
		IN_ClosingRampValue : REAL;
		IN_OutMin : REAL; (*Min Opening [%]*)
		IN_OutMax : REAL; (*Max Opening [%]*)
		IN_HMIAutoForce : BOOL;
		IN_ManEn : BOOL;
		IN_MaskEn : BOOL;
		IN_Reset : BOOL; (*Fault Reset*)
	END_VAR
	VAR_OUTPUT
		OUT_Cv : REAL; (*Analog output (0.0 - 100.0)*)
		OUT_Alarm : BOOL; (*Falt Output for Alarm*)
		OUT_RampDone : BOOL; (*Ramp Done*)
		OUT_FBKFault : BOOL;
		OUT_FBK : REAL; (*Analog Input FeedBack Value 0.0 - 100.0%*)
	END_VAR
	VAR_IN_OUT
		IO : IO_Valve_Mod_Type;
		HMI : HMI_Valve_Mod_Type;
	END_VAR
	VAR
		VAR_Fault : BOOL; (*Falt Output for Alarm*)
		VAR_iFault : BOOL;
		VAR_ConfigPosition : BOOL;
		VAR_OutMan : REAL;
		VAR_Open : REAL;
		VAR_iOpen : REAL;
		TMR_TOF_DOValveOn : TOF;
		VAR_FirstCycle : BOOL;
		VAR_DOValveOn : BOOL;
		VAR_DOValveOff : BOOL;
		VAR_DIFeedBackOpen : BOOL;
		VAR_DIFeedBackClose : BOOL;
		VAR_Mask : BOOL;
		TMR_TON_PositionFiltered : TON;
		VAR_ManOn : BOOL;
		VAR_Auto : BOOL;
		LCRMovingRamp : LCRRamp;
		VAR_OpeningRamp : REAL;
		VAR_ClosingRamp : REAL;
		LCRLimScal_AO : LCRLimScal;
		LCRLimScal_AI : LCRLimScal;
		VAR_FaultSensorOn : BOOL;
		VAR_FaultSensorOff : BOOL;
		VAR_FaultSensorFBK : BOOL;
	END_VAR
END_FUNCTION_BLOCK

FUNCTION_BLOCK Fan_Obj
	VAR_INPUT
		IN_ConfigPresent : BOOL;
		IN_RoofType : BOOL; (*0: Fan 1: Galvani*)
		IN_GalvaniRoofFlowSet : BOOL;
		IN_CgfHmiLampOn : BOOL;
		IN_FanNumber : USINT := 1;
		IN_AutoSpeed : REAL;
		IN_Enable : BOOL;
		IN_HMIAutoForce : BOOL;
		IN_Reset : BOOL; (*Control: Alarm Reset Push Button*)
	END_VAR
	VAR_OUTPUT
		OUT_Alarm : BOOL;
		Out_Light : BOOL; (*v4.A.A.1.7.0*)
		OUT_OverloadFault : BOOL;
	END_VAR
	VAR_IN_OUT
		IO : IO_FanMain_Type;
		HMI : HMI_Fan_Type;
		ALARM : FanZoneAlarm_Type;
	END_VAR
	VAR
		TMR_TON_OnDelay : ARRAY[1..6] OF TON;
		TMR_TON_OffDelay : ARRAY[1..6] OF TON;
		VAR_Auto : ARRAY[1..6] OF BOOL;
		TMR_TON_OnDelay_Gal : TON;
		TMR_TON_OffDelay_Gal : TON;
		VAR_Auto_Gal : BOOL;
		VAR_OUT : REAL;
		VAR_GalvaniOn : BOOL;
		VAR_GalvaniFlowSet : BOOL;
		VAR_AbsoluteFilter : BOOL;
		VAR_PreFilter : BOOL;
		VAR_PressurizedOnAlarm : BOOL;
		VAR_ResetHMI : BOOL;
		VAR_i : USINT;
	END_VAR
END_FUNCTION_BLOCK

FUNCTION_BLOCK MotionFan_Obj
	VAR_INPUT
		IN_ConfigPresent : BOOL;
		IN_Enable : BOOL; (*Safety OK ( True if not used)*)
		IN_AutoCnd : BOOL; (*Automation Logic Input*)
		IN_Reset : BOOL; (*Fault Reset*)
		IN_FBKDelay : TIME := T#500ms; (*Time: Running Control Delay*)
	END_VAR
	VAR_OUTPUT
		OUT_Running : BOOL; (*Motor On*)
		OUT_IsolatedFault : BOOL;
		OUT_ContactorFBKFault : BOOL;
		OUT_OverloadFault : BOOL;
		OUT_Alarm : BOOL; (*Output for Alarm*)
	END_VAR
	VAR_IN_OUT
		IO : IO_MotionFan_Type;
	END_VAR
	VAR
		TMR_TOF : TON;
		TMR_TON : TON;
		VAR_ContactorFBK : BOOL;
		VAR_Isolated : BOOL;
		VAR_Overload : BOOL;
		VAR_Fault : BOOL; (*Alarm Output for Fault or Warning*)
	END_VAR
END_FUNCTION_BLOCK
(*Shift Register Object*)

FUNCTION_BLOCK CapPhotoCell_SftObj_old (* *) (*$GROUP=User,$CAT=User,$GROUPICON=User.png,$CATICON=User.png*)
	VAR_INPUT
		IN_ConfigPresent : BOOL; (*Configuration: Device Present*)
		IN_Enable : BOOL; (*Configuration: Enable *)
		IN_Alarm : BOOL; (*Configuration: Timeout Alarm Control Enable*)
		IN_WaitOn : BOOL; (*Control: On State Wait Request*)
		IN_WaitOff : BOOL; (*Control: Off State Wait Request*)
		IN_MachinePitch : BOOL; (*Control: Machine Pitch Pulse*)
		IN_ResetCounters : BOOL;
		IN_MaskEn : BOOL; (*Control: Mask Enable*)
		IN_GrippersNumber : USINT; (*Control : Grip Number For Repetitive Control*)
		IN_CBlockAbsoluteValue : USINT; (*Control: Container Stop Threshold For Absolute Container Lack*)
		IN_CBlockRepetitiveValue : USINT; (*Control: Container Stop Threshold For Repetitive Container Lack*)
		IN_MStopAbsoluteValue : USINT; (*Control: Critical Stop Threshold For Absolute Container Lack*)
		IN_MStopConsecutiveValue : USINT; (*Control: Critical Stop Threshold For Consecutive Container Lack*)
	END_VAR
	VAR_OUTPUT
		OUT : BOOL; (*State Switching Delayed*)
		OUT_CBlockRepetitive : BOOL; (*Container Stop For Repetitive Lack Errors*)
		OUT_CBlockAbsolute : BOOL; (*Container Stop For Absolute Lack Errors*)
		OUT_MStopConsecutive : BOOL; (*Critical Stop For Consecutive*)
		OUT_MStopAbsolute : BOOL; (*Critical Stop For Absolute*)
		OUT_AlwaysTrueError : BOOL;
	END_VAR
	VAR_IN_OUT
		IO : IO_Digital_IN_Type; (*State: Digital Input Structure*)
		HMI : HMI_Photocell_Type;
		SHIFT_Position : UINT;
	END_VAR
	VAR CONSTANT
		CST_AlwaysTrueMaxSteps : USINT := 10; (*Max Number Of Steps With The Photocell Always TRUE*)
		CST_RepetitiveArrayDim : USINT := 50; (*Repetitive Array Dimension*)
	END_VAR
	VAR
		TMR_TON_TotalCounterReset : TON;
		VAR_Mask : BOOL;
		VAR_Signal : BOOL;
		VAR_CounterResetMemory : BOOL;
		VAR_TotalCounterResetMemory : BOOL;
		VAR_EdgeChecked : BOOL;
		VAR_GrippersNumber : USINT;
		VAR_ActualValveCounter : USINT := 1;
		VAR_RepetitiveCounterArray : ARRAY[1..CST_RepetitiveArrayDim] OF USINT;
	END_VAR
END_FUNCTION_BLOCK

FUNCTION_BLOCK CapPhotoCell_SftObj (* *) (*$GROUP=User,$CAT=User,$GROUPICON=User.png,$CATICON=User.png*)
	VAR_INPUT
		IN_ConfigPresent : BOOL; (*Configuration: Device Present*)
		IN_Enable : BOOL; (*Configuration: Enable *)
		IN_Alarm : BOOL; (*Configuration: Timeout Alarm Control Enable*)
		IN_WaitOn : BOOL; (*Control: On State Wait Request*)
		IN_WaitOff : BOOL; (*Control: Off State Wait Request*)
		IN_MachinePitch : BOOL; (*Control: Machine Pitch Pulse*)
		IN_ResetCounters : BOOL; (*V1.61 Reset Absolute Errors*)
		IN_ResetCountersConsecutive : BOOL; (*V1.61 Reset Consecutive errors*)
		IN_MaskEn : BOOL; (*Control: Mask Enable*)
		IN_GrippersNumber : USINT; (*Control : Grip Number For Repetitive Control*)
		IN_CBlockAbsoluteValue : USINT; (*Control: Container Stop Threshold For Absolute Container Lack*)
		IN_CBlockAbsoluteQuantity : UINT; (*Control: Critical Stop Threshold For Consecutive Container Lack*)
		IN_CBlockRepetitiveValue : USINT; (*Control: Container Stop Threshold For Repetitive Container Lack*)
		IN_MStopConsecutiveValue : USINT; (*Control: Critical Stop Threshold For Consecutive Container Lack*)
	END_VAR
	VAR_OUTPUT
		OUT : BOOL; (*State Switching Delayed*)
		OUT_CBlockRepetitive : BOOL; (*Container Stop For Repetitive Lack Errors*)
		OUT_CBlockAbsolute : BOOL; (*Container Stop For Absolute Lack Errors*)
		OUT_MStopConsecutive : BOOL; (*Critical Stop For Consecutive*)
		OUT_AlwaysTrueError : BOOL;
	END_VAR
	VAR_IN_OUT
		IO : IO_Digital_IN_Type; (*State: Digital Input Structure*)
		HMI : HMI_Photocell_Type;
		SHIFT_Position : UINT;
	END_VAR
	VAR CONSTANT
		CST_AlwaysTrueMaxSteps : USINT := 10; (*Max Number Of Steps With The Photocell Always TRUE*)
		CST_CounterArrayDim : USINT := 50; (*Repetitive Array Dimension*)
	END_VAR
	VAR
		TMR_TON_TotalCounterReset : TON;
		VAR_AbsoluteErrorN : USINT := 1;
		VAR_Mask : BOOL;
		VAR_Signal : BOOL;
		VAR_CounterResetMemory : BOOL;
		VAR_CounterConsResetMemory : BOOL; (*V1.61*)
		VAR_TotalCounterResetMemory : BOOL;
		VAR_EdgeChecked : BOOL;
		VAR_GrippersNumber : USINT;
		VAR_ActualValveCounter : USINT := 1;
		VAR_i : USINT;
		VAR_CapsReleased : UDINT;
		VAR_AbsoluteCounterArray : ARRAY[1..CST_CounterArrayDim] OF UDINT;
		VAR_RepetitiveCounterArray : ARRAY[1..CST_CounterArrayDim] OF USINT;
	END_VAR
END_FUNCTION_BLOCK

FUNCTION_BLOCK Ejector_SftObj (* Container Ejector Valve *)
	VAR_INPUT
		IN_ConfigPresent : BOOL; (*Configuration: Device Present*)
		IN_ConfigType : BOOL; (*Configuration: Device Type (0: Monostable - 1: Bistable)*)
		IN_Enable : BOOL;
		IN_MachinePitch : BOOL;
		IN_FillingErrorEject : BOOL;
		IN_SamplingModeActive : BOOL; (*V1.61*)
		IN_ResetCounters : BOOL;
		IN_HMIAutoForce : BOOL;
		IN_ManEn : BOOL;
		IN_MaskEn : BOOL;
		IN_ShiftPosition : UINT;
		IN_CBlockAbsoluteValue : USINT; (*Control: Container Stop Threshold For Absolute Container Lack*)
		IN_MStopConsecutiveValue : USINT; (*Control: Machine Stop Threshold For Consecutive Container Lack*)
	END_VAR
	VAR_OUTPUT
		OUT : BOOL; (*Stroke done*)
		OUT_CBlockAbsolute : BOOL; (*Container Stop For Absolute Lack Errors*)
		OUT_MStopConsecutive : BOOL; (*Critical Stop For Consecutive*)
	END_VAR
	VAR_IN_OUT
		IO : IO_Valve_Type;
		HMI : HMI_Valve_Ejector_Type;
	END_VAR
	VAR
		TMR_TON_TotalCounterReset : TON;
		VAR_Mask : BOOL;
		VAR_ManOn : BOOL;
		VAR_Auto : BOOL;
		VAR_AutoCnd : BOOL;
		VAR_CounterResetMemory : BOOL;
		VAR_TotalCounterResetMemory : BOOL;
		VAR_ValveOpened : BOOL;
		VAR_ValveClosed : BOOL;
	END_VAR
END_FUNCTION_BLOCK

FUNCTION_BLOCK PhotoCell_SftObj (* *) (*$GROUP=User,$CAT=User,$GROUPICON=User.png,$CATICON=User.png*)
	VAR_INPUT
		IN_ConfigPresent : BOOL; (*Configuration: Device Present*)
		IN_Enable : BOOL; (*Configuration: Enable *)
		IN_Alarm : BOOL; (*Configuration: Alarm Control Enable*)
		IN_WaitOn : BOOL; (*Control: On State Wait Request*)
		IN_WaitOff : BOOL; (*Control: Off State Wait Request*)
		IN_MachinePitch : BOOL; (*Control: Machine Pitch Pulse*)
		IN_ResetCounters : BOOL;
		IN_WritePresenceEnable : BOOL; (*Configuration Type of Photocell (0: Disabel Write Presence, 1: Enable Write Presence)*)
		IN_MaskEn : BOOL; (*Control: Mask Enable*)
		IN_GrippersNumber : USINT; (*Control : Grip Number For Repetitive Control*)
		IN_CBlockAbsoluteValue : USINT; (*Control: Container Stop Threshold For Absolute Container Lack*)
		IN_CBlockRepetitiveValue : USINT; (*Control: Container Stop Threshold For Repetitive Container Lack*)
		IN_MStopAbsoluteValue : USINT; (*Control: Machine Stop Threshold For Absolute Container Lack*)
		IN_MStopConsecutiveValue : USINT; (*Control: Machine Stop Threshold For Consecutive Container Lack*)
	END_VAR
	VAR_OUTPUT
		OUT : BOOL; (*State Switching Delayed*)
		OUT_CBlockRepetitive : BOOL; (*Container Stop For Repetitive Lack Errors*)
		OUT_CBlockAbsolute : BOOL; (*Container Stop For Absolute Lack Errors*)
		OUT_MStopConsecutive : BOOL; (*Critical Stop For Consecutive*)
		OUT_MStopAbsolute : BOOL; (*Critical Stop For Absolute*)
		OUT_AlwaysTrueError : BOOL;
	END_VAR
	VAR_IN_OUT
		IO : IO_Digital_IN_Type; (*State: Digital Input Structure*)
		HMI : HMI_Photocell_Type;
		SHIFT_Position : UINT;
	END_VAR
	VAR CONSTANT
		CST_AlwaysTrueMaxSteps : USINT := 10; (*Max Number Of Steps With The Photocell Always TRUE*)
		CST_RepetitiveArrayDim : USINT := 50; (*Repetitive Array Dimension*)
	END_VAR
	VAR
		TMR_TON_TotalCounterReset : TON;
		VAR_Mask : BOOL;
		VAR_Signal : BOOL;
		VAR_CounterResetMemory : BOOL;
		VAR_TotalCounterResetMemory : BOOL;
		VAR_EdgeChecked : BOOL;
		VAR_GrippersNumber : USINT;
		VAR_ActualValveCounter : USINT := 1;
		VAR_RepetitiveCounterArray : ARRAY[1..CST_RepetitiveArrayDim] OF USINT;
	END_VAR
END_FUNCTION_BLOCK

(* ---- UVtronic_Std.st ---- *)
FUNCTION_BLOCK UVtronic_Std
	IF NOT VAR_FirstCycle THEN
		HMI.ManOff		:= FALSE;
		HMI.ManOn		:= FALSE;
		VAR_FirstCycle	:= TRUE;
	END_IF

	IF IN_ConfigPresent THEN
		(*****************************************************************)
		(*****************************START*******************************)
		(*****************************************************************)
		IF (EDGENEG(IN_ManEn) AND HMI.ManOn) OR IN_HMIAutoForce THEN
			HMI.ManOn	:= FALSE;
			HMI.ManOff	:= FALSE;
		END_IF

		VAR_Mask := HMI.Mask AND IN_MaskEn;
		VAR_Auto := NOT HMI.ManOff AND NOT HMI.ManOn;

		IF VAR_Fault OR NOT IN_Enable THEN
			IO.DO_MotorON := FALSE;
		ELSIF VAR_Auto THEN
			IO.DO_MotorON := IN_AutoCnd;
		ELSE
			IO.DO_MotorON := HMI.ManOn;
		END_IF

		(*****************************************************************)
		(**************************ALARM LOGIC****************************)
		(*****************************************************************)
		TMR_TON(IN := IO.DO_MotorON,
				PT := IN_FBKDelay);

		TMR_TOF(IN := NOT IO.DO_MotorON,
				PT := IN_FBKDelay);

		IF IN_Reset THEN
			VAR_ContactorFBK	:= FALSE;
			VAR_GeneralFault	:= FALSE;
			VAR_Overload		:= FALSE;
			VAR_NotReady		:= FALSE;
		END_IF

		IF ((TMR_TON.Q AND IO.DI_ContactorFBK) OR (TMR_TOF.Q AND NOT IO.DI_ContactorFBK)) AND NOT IN_ConfigType AND NOT VAR_Mask THEN
			VAR_ContactorFBK := NOT IN_Simulation;
		END_IF

		IF IO.DI_GeneralFault AND NOT VAR_Mask THEN
			VAR_GeneralFault := NOT IN_Simulation;
		END_IF

		IF NOT IO.DI_OverloadOK AND NOT IN_ConfigType AND NOT VAR_Mask THEN
			VAR_Overload := NOT IN_Simulation;
		END_IF

		IF NOT IO.DI_Ready AND NOT VAR_Mask THEN
			VAR_NotReady := NOT IN_Simulation;
		END_IF

		VAR_Fault := (VAR_ContactorFBK OR VAR_GeneralFault OR VAR_Overload OR VAR_NotReady AND IN_Enable) AND NOT IN_Simulation;

		(*****************************************************************)
		(******************************HMI********************************)
		(*****************************************************************)
		HMI.Out				:= IO.DO_MotorON;
		HMI.Alarm			:= VAR_Fault;
		HMI.Isolated		:= FALSE;
		HMI.Overload		:= VAR_Overload;
		HMI.FeedBack		:= VAR_ContactorFBK;
		HMI.ConfigPresent	:= IN_ConfigPresent;
		HMI.ManEnable		:= IN_ManEn;
		HMI.MaskEnable		:= IN_MaskEn;

		(*****************************************************************)
		(******************************OUT********************************)
		(*****************************************************************)
		OUT_Running				:= IO.DO_MotorON;
		OUT_NotReady			:= VAR_NotReady;
		OUT_GeneralFault		:= VAR_GeneralFault;
		OUT_ContactorFBKFault	:= VAR_ContactorFBK;
		OUT_OverloadFault		:= VAR_Overload;
		OUT_Alarm				:= VAR_Fault;
	ELSE
		memset(ADR(HMI), 0, SIZEOF(HMI));
		OUT_Running				:= FALSE;
		OUT_NotReady			:= FALSE;
		OUT_GeneralFault		:= FALSE;
		OUT_ContactorFBKFault	:= FALSE;
		OUT_OverloadFault		:= FALSE;
		OUT_Alarm				:= FALSE;
		IO.DO_MotorON			:= FALSE;
	END_IF
END_FUNCTION_BLOCK

(* ---- Valve_Dig.st ---- *)
FUNCTION_BLOCK Valve_Dig
	IF NOT IN_Simulation AND IN_ConfigPositionSensorOpened AND IN_ConfigPositionSensorClosed AND NOT VAR_Mask THEN
		TMR_TOF_FeedBackOpen.IN 	:= IO.DI_Opened;
		VAR_FeedBackOpen			:= TMR_TOF_FeedBackOpen.Q;
		TMR_TOF_FeedBackClose.IN	:= IO.DI_Closed;
		VAR_FeedBackClose			:= TMR_TOF_FeedBackClose.Q;
	ELSIF NOT IN_Simulation AND IN_ConfigPositionSensorOpened AND NOT IN_ConfigPositionSensorClosed AND NOT VAR_Mask THEN
		TMR_TOF_FeedBackOpen.IN 	:= IO.DI_Opened;
		VAR_FeedBackOpen			:= TMR_TOF_FeedBackOpen.Q;
		TMR_TOF_FeedBackClose.IN	:= NOT IO.DI_Opened;
		VAR_FeedBackClose			:= TMR_TOF_FeedBackClose.Q;
	ELSIF NOT IN_Simulation AND NOT IN_ConfigPositionSensorOpened AND IN_ConfigPositionSensorClosed AND NOT VAR_Mask THEN
		TMR_TOF_FeedBackOpen.IN 	:= NOT IO.DI_Closed;
		VAR_FeedBackOpen			:= TMR_TOF_FeedBackOpen.Q;
		TMR_TOF_FeedBackClose.IN	:= IO.DI_Closed;
		VAR_FeedBackClose			:= TMR_TOF_FeedBackClose.Q;
	ELSE
		TMR_TOF_FeedBackOpen.IN 	:= VAR_ValveOpened;
		VAR_FeedBackOpen			:= TMR_TOF_FeedBackOpen.Q;
		TMR_TOF_FeedBackClose.IN	:= NOT VAR_ValveOpened;
		VAR_FeedBackClose			:= TMR_TOF_FeedBackClose.Q;
	END_IF

	TMR_TOF_FeedBackOpen.PT		:= t#50ms;
	TMR_TOF_FeedBackOpen();
	TMR_TOF_FeedBackClose.PT	:= t#50ms;
	TMR_TOF_FeedBackClose();

	IF NOT IN_Simulation THEN
		VAR_Enable	:= IN_Enable;
		VAR_iFault	:= VAR_Fault;
		VAR_Mask	:= HMI.Mask AND IN_MaskEn;
	ELSE
		VAR_Enable	:= TRUE;
		VAR_iFault	:= HMI.Mask;
		VAR_Mask	:= FALSE;
	END_IF

	(* Local *)
	IF IN_ManEn AND NOT IN_HMIAutoForce THEN
		VAR_ManOn	:= HMI.ManOn;
		VAR_Auto	:= NOT HMI.ManOff AND NOT HMI.ManOn;
	ELSE
		VAR_ManOn	:= FALSE;
		VAR_Auto	:= TRUE;
		HMI.ManOn	:= FALSE;
		HMI.ManOff	:= FALSE;
	END_IF

	VAR_ConfigPosition	:= (IN_ConfigPositionSensorOpened OR IN_ConfigPositionSensorClosed) AND IN_MaskEn;
	VAR_AutoCnd := (IN_AutoCnd AND (IN_Cnd OR NOT IN_EnableCnd)) OR (IN_FlipRequest AND NOT OUT_FlipDone AND IN_FlipEnable);

	TMR_TON_Flip(	IN  := IN_FlipRequest,
					PT  := MIN(IN_FlipTime, MAX_Flip_Time));

	IF IN_FlipEnable THEN
		OUT_FlipDone := TMR_TON_Flip.Q;
	ELSE
		OUT_FlipDone := IN_FlipRequest;
	END_IF

	IF IN_ConfigPresent THEN
		IF IN_ConfigType THEN
			IF VAR_Enable THEN
				IF VAR_Auto THEN
					VAR_ValveOpened := VAR_AutoCnd;
				ELSIF VAR_ManOn THEN
					VAR_ValveOpened := TRUE;
				ELSE
					VAR_ValveOpened := FALSE;
				END_IF
				VAR_ValveClosed := NOT VAR_ValveOpened;
			ELSE
				VAR_ValveOpened := FALSE;
				VAR_ValveClosed := FALSE;
			END_IF
		ELSE
			IF VAR_Enable THEN
				IF VAR_Auto THEN
					VAR_ValveOpened := VAR_AutoCnd;
				ELSIF VAR_ManOn THEN
					VAR_ValveOpened := TRUE;
				ELSE
					VAR_ValveOpened := FALSE;
				END_IF
			ELSE
				VAR_ValveOpened := FALSE;
			END_IF
			VAR_ValveClosed := NOT VAR_ValveOpened;
		END_IF

		(*********************** Alarm Logic ************************)
		TMR_TON_ControlEnableDelay(	IN := IN_ConfigPositionSensorOpened OR IN_ConfigPositionSensorClosed,
									PT := t#300ms);

		IF TMR_TON_ControlEnableDelay.Q THEN
			TMR_TON_Opened  (IN := VAR_ValveOpened, PT := IN_StrokeTime);
			TMR_TON_Closed	(IN := VAR_ValveClosed, PT := IN_StrokeTime);
			IF TMR_TON_Closed.Q AND (VAR_FeedBackOpen OR NOT VAR_FeedBackClose) THEN
				VAR_Fault := TRUE;
			ELSIF TMR_TON_Opened.Q AND (NOT VAR_FeedBackOpen OR VAR_FeedBackClose) THEN
				VAR_Fault := TRUE;
			ELSIF IN_Reset THEN
				VAR_Fault := FALSE;
			END_IF
		ELSIF IN_Reset THEN
			VAR_Fault := FALSE;
		END_IF

		OUT_Alarm := VAR_iFault;

		TMR_TON_ClosedFilter.IN := VAR_FeedBackClose AND NOT VAR_FeedBackOpen;
		TMR_TON_ClosedFilter.PT := T#500ms;
		TMR_TON_ClosedFilter();

		OUT_ClosedFiltered := TMR_TON_ClosedFilter.Q;

		TMR_TON_OpenedFilter.IN := NOT VAR_FeedBackClose AND VAR_FeedBackOpen;
		TMR_TON_OpenedFilter.PT := T#500ms;
		TMR_TON_OpenedFilter();

		OUT_OpenedFiltered 	:= TMR_TON_OpenedFilter.Q;
	 	OUT					:= VAR_ValveOpened;
	ELSE
		OUT_Alarm				:= FALSE;
		OUT_ClosedFiltered		:= NOT VAR_AutoCnd;
		OUT_OpenedFiltered		:= VAR_AutoCnd;
		OUT						:= VAR_AutoCnd;
		VAR_ValveOpened			:= FALSE;
		VAR_ValveClosed			:= FALSE;
		VAR_iFault				:= FALSE;
	END_IF

	(* HMI *)
	HMI.ManEnable		:= IN_ManEn;
	HMI.ConfigPresent	:= IN_ConfigPresent;
	HMI.ConfigPosition	:= VAR_ConfigPosition;
	HMI.MaskEnable		:= IN_MaskEn;
	HMI.Alarm			:= VAR_iFault;

	IF IN_ConfigNormallyOpen THEN //v1.5
		HMI.Opened			:= OUT_ClosedFiltered; //v1.5
		HMI.Closed			:= OUT_OpenedFiltered; //v1.5
	ELSE
		HMI.Opened			:= OUT_OpenedFiltered;
		HMI.Closed			:= OUT_ClosedFiltered;
	END_IF //v1.5

	(* IO *)
	IF NOT IN_Simulation THEN
		IO.DO_Opened	:= VAR_ValveOpened;
		IO.DO_Closed	:= VAR_ValveClosed;
		HMI.Out			:= IO.DO_Opened;
	ELSE
		IO.DO_Opened	:= FALSE;
		IO.DO_Closed	:= FALSE;
		HMI.Out			:= VAR_ValveOpened;
	END_IF
END_FUNCTION_BLOCK

(* ---- Valve_Dig_Mac.st ---- *)
FUNCTION_BLOCK Valve_Dig_Mac
	IF NOT IN_Simulation AND IN_ConfigPositionSensorOpened AND IN_ConfigPositionSensorClosed AND NOT VAR_Mask THEN
		TMR_TOF_FeedBackOpen.IN 	:= IO.DI_Opened;
		VAR_FeedBackOpen			:= TMR_TOF_FeedBackOpen.Q;
		TMR_TOF_FeedBackClose.IN	:= IO.DI_Closed;
		VAR_FeedBackClose			:= TMR_TOF_FeedBackClose.Q;
	ELSIF NOT IN_Simulation AND IN_ConfigPositionSensorOpened AND NOT IN_ConfigPositionSensorClosed AND NOT VAR_Mask THEN
		TMR_TOF_FeedBackOpen.IN 	:= IO.DI_Opened;
		VAR_FeedBackOpen			:= TMR_TOF_FeedBackOpen.Q;
		TMR_TOF_FeedBackClose.IN	:= NOT IO.DO_Closed;
		VAR_FeedBackClose			:= TMR_TOF_FeedBackClose.Q;
	ELSIF NOT IN_Simulation AND NOT IN_ConfigPositionSensorOpened AND IN_ConfigPositionSensorClosed AND NOT VAR_Mask THEN
		TMR_TOF_FeedBackOpen.IN 	:= NOT IO.DI_Closed;
		VAR_FeedBackOpen			:= TMR_TOF_FeedBackOpen.Q;
		TMR_TOF_FeedBackClose.IN	:= IO.DI_Closed;
		VAR_FeedBackClose			:= TMR_TOF_FeedBackClose.Q;
	ELSE
		TMR_TOF_FeedBackOpen.IN 	:= VAR_ValveOpened;
		VAR_FeedBackOpen			:= TMR_TOF_FeedBackOpen.Q;
		TMR_TOF_FeedBackClose.IN	:= NOT VAR_ValveOpened;
		VAR_FeedBackClose			:= TMR_TOF_FeedBackClose.Q;
	END_IF

	TMR_TOF_FeedBackOpen.PT		:= t#50ms;
	TMR_TOF_FeedBackOpen();
	TMR_TOF_FeedBackClose.PT	:= t#50ms;
	TMR_TOF_FeedBackClose();

	IF NOT IN_Simulation THEN
		VAR_Enable	:= IN_Enable;
		VAR_iFault	:= VAR_Fault;
		VAR_Mask	:= HMI.Mask AND IN_MaskEn;
	ELSE
		VAR_Enable	:= TRUE;
		VAR_iFault	:= HMI.Mask;
		VAR_Mask	:= FALSE;
	END_IF

	(* Local *)
	IF IN_ManEn AND NOT IN_HMIAutoForce THEN
		VAR_ManOn	:= HMI.ManOn;
		VAR_Auto	:= NOT HMI.ManOff AND NOT HMI.ManOn;
	ELSE
		VAR_ManOn	:= FALSE;
		VAR_Auto	:= TRUE;
		HMI.ManOn	:= FALSE;
		HMI.ManOff	:= FALSE;
	END_IF

	VAR_ConfigPosition	:= (IN_ConfigPositionSensorOpened OR IN_ConfigPositionSensorClosed) AND IN_MaskEn;
	VAR_AutoCnd := (IN_AutoCnd AND (IN_Cnd OR NOT IN_EnableCnd)) OR (IN_FlipRequest AND NOT OUT_FlipDone AND IN_FlipEnable);

	TMR_TON_Flip(	IN  := IN_FlipRequest,
					PT  := MIN(IN_FlipTime, MAX_Flip_Time));

	IF IN_FlipEnable THEN
		OUT_FlipDone := TMR_TON_Flip.Q;
	ELSE
		OUT_FlipDone := IN_FlipRequest;
	END_IF

	IF IN_ConfigPresent THEN
		IF IN_ConfigType THEN
			IF VAR_Enable THEN
				IF VAR_Auto THEN
					VAR_ValveOpened := VAR_AutoCnd;
				ELSIF VAR_ManOn THEN
					VAR_ValveOpened := TRUE;
				ELSE
					VAR_ValveOpened := FALSE;
				END_IF
				VAR_ValveClosed := NOT VAR_ValveOpened;
			ELSE
				VAR_ValveOpened := FALSE;
				VAR_ValveClosed := FALSE;
			END_IF
		ELSE
			IF VAR_Enable THEN
				IF VAR_Auto THEN
					VAR_ValveOpened := VAR_AutoCnd;
				ELSIF VAR_ManOn THEN
					VAR_ValveOpened := TRUE;
				ELSE
					VAR_ValveOpened := FALSE;
				END_IF
			ELSE
				VAR_ValveOpened := FALSE;
			END_IF
			VAR_ValveClosed := NOT VAR_ValveOpened;
		END_IF

		(*********************** Alarm Logic ************************)
		TMR_TON_ControlEnableDelay(	IN := IN_ConfigPositionSensorOpened OR IN_ConfigPositionSensorClosed,
									PT := t#300ms);

		IF TMR_TON_ControlEnableDelay.Q THEN
			TMR_TON_Opened  (IN := VAR_ValveOpened, PT := IN_StrokeTime);
			TMR_TON_Closed	(IN := VAR_ValveClosed, PT := IN_StrokeTime);
			IF TMR_TON_Closed.Q AND (VAR_FeedBackOpen OR NOT VAR_FeedBackClose) THEN
				VAR_Fault := TRUE;
			ELSIF TMR_TON_Opened.Q AND (NOT VAR_FeedBackOpen OR VAR_FeedBackClose) THEN
				VAR_Fault := TRUE;
			ELSIF IN_Reset THEN
				VAR_Fault := FALSE;
			END_IF
		ELSIF IN_Reset THEN
			VAR_Fault := FALSE;
		END_IF

		OUT_Alarm := VAR_iFault;

		IF IN_ConfigPositionSensorOpened THEN
			TMR_TON_ClosedFilter.IN := VAR_FeedBackClose AND NOT VAR_FeedBackOpen;
			TMR_TON_ClosedFilter.PT := T#500ms;
		ELSE
			TMR_TON_ClosedFilter.IN := VAR_ValveClosed;
			TMR_TON_ClosedFilter.PT := T#1s;
		END_IF

		TMR_TON_ClosedFilter();

		OUT_ClosedFiltered := TMR_TON_ClosedFilter.Q;

		IF IN_ConfigPositionSensorClosed THEN
			TMR_TON_OpenedFilter.IN := NOT VAR_FeedBackClose AND VAR_FeedBackOpen;
			TMR_TON_OpenedFilter.PT := T#500ms;
		ELSE
			TMR_TON_OpenedFilter.IN := VAR_ValveOpened;
			TMR_TON_OpenedFilter.PT := T#1s;
		END_IF
		TMR_TON_OpenedFilter();

		OUT_OpenedFiltered := TMR_TON_OpenedFilter.Q;
	 	OUT	:= VAR_ValveOpened;
	ELSE
		OUT_Alarm				:= FALSE;
		OUT_ClosedFiltered		:= NOT VAR_AutoCnd;
		OUT_OpenedFiltered		:= VAR_AutoCnd;
		OUT						:= VAR_AutoCnd;
		VAR_ValveOpened			:= FALSE;
		VAR_ValveClosed			:= FALSE;
	END_IF

	(* HMI *)
	HMI.ManEnable		:= IN_ManEn;
	HMI.ConfigPresent	:= IN_ConfigPresent;
	HMI.ConfigPosition	:= VAR_ConfigPosition;
	HMI.MaskEnable		:= IN_MaskEn;
	HMI.Alarm			:= VAR_iFault;
	HMI.Opened			:= OUT_OpenedFiltered;
	HMI.Closed			:= OUT_ClosedFiltered;

	(* IO *)
	TMR_TP_Block.IN		:= VAR_ValveClosed;
	TMR_TP_Block.PT		:= t#3s;
	TMR_TP_Block.RESET	:= NOT VAR_ValveClosed;
	TMR_TP_Block();

	TMR_TP_Release.IN	:= VAR_ValveOpened;
	TMR_TP_Release.PT	:= t#3s;
	TMR_TP_Release.RESET:= NOT VAR_ValveOpened;
	TMR_TP_Release();

	IF NOT IN_Simulation THEN
		IO.DO_Opened	:= TMR_TP_Release.Q;
		IO.DO_Closed	:= TMR_TP_Block.Q;
		HMI.Out			:= VAR_ValveOpened;
	ELSE
		IO.DO_Opened	:= FALSE;
		IO.DO_Closed	:= FALSE;
		HMI.Out			:= VAR_ValveOpened;
	END_IF
END_FUNCTION_BLOCK

(* ---- Valve_Mod.st ---- *)
FUNCTION_BLOCK Valve_Mod
	IF NOT VAR_FirstCycle THEN
		memset(ADR(HMI),0,SIZEOF(HMI));
		HMI.ManOff		:= FALSE;
		HMI.ManOn		:= FALSE;
		VAR_FirstCycle	:= TRUE;
	END_IF

	(*IO*)
	IF NOT IN_Simulation AND IN_ConfigPositionSensorOpened AND IN_ConfigPositionSensorClosed THEN
		VAR_DIFeedBackOpen	:= IO.Valve.DI_Opened;
		VAR_DIFeedBackClose	:= IO.Valve.DI_Closed;
	ELSIF NOT IN_Simulation AND IN_ConfigPositionSensorOpened AND NOT IN_ConfigPositionSensorClosed THEN
		VAR_DIFeedBackOpen	:= IO.Valve.DI_Opened;
		VAR_DIFeedBackClose	:= NOT IO.Valve.DI_Opened;
	ELSIF NOT IN_Simulation AND NOT IN_ConfigPositionSensorOpened AND IN_ConfigPositionSensorClosed THEN
		VAR_DIFeedBackOpen	:= NOT IO.Valve.DI_Closed;
		VAR_DIFeedBackClose	:= IO.Valve.DI_Closed;
	ELSE
		VAR_DIFeedBackOpen	:= VAR_DOValveOn;
		VAR_DIFeedBackClose	:= VAR_DOValveOff;
	END_IF

	IF NOT IN_Simulation THEN
		VAR_iFault			:= VAR_Fault;
		VAR_Mask 			:= HMI.Mask AND IN_MaskEn;
	ELSE
		VAR_iFault			:= HMI.Mask;
		VAR_Mask 			:= FALSE;
	END_IF

	(*Local*)
	IF IN_HMIAutoForce OR NOT IN_ManEn THEN
		HMI.ManOn	:= FALSE;
		HMI.ManOff	:= FALSE;
	END_IF

	VAR_ManOn 			:= HMI.ManOn;
	VAR_Auto			:= NOT HMI.ManOff AND NOT HMI.ManOn;
	VAR_OutMan			:= HMI.OUT_Man;
	VAR_ConfigPosition	:= IN_ConfigPositionSensorOpened OR IN_ConfigPositionSensorClosed;

	IF IN_ConfigPresent THEN
		IF IN_Enable THEN
			IF VAR_Auto AND IN_AutoCnd THEN
				VAR_iOpen := IN_AutoVal;
			ELSIF VAR_ManOn THEN
				VAR_iOpen := VAR_OutMan;
			ELSE
				VAR_iOpen := 0.0;
			END_IF
		ELSE
			VAR_iOpen := 0.0;
		END_IF

		(*****************************************************************)
		(****************************FAULTS*******************************)
		(*****************************************************************)
		IF IN_ConfigPositionSensorOpened THEN
			IF ((VAR_Open = 0.0) AND (VAR_DIFeedBackOpen) OR (VAR_Open = 100.0) AND (NOT VAR_DIFeedBackOpen)) THEN
				VAR_FaultSensorOn := TRUE;
			ELSE
				VAR_FaultSensorOn := FALSE;
			END_IF
		ELSE
			VAR_FaultSensorOn := FALSE;
		END_IF

		IF IN_ConfigPositionSensorClosed THEN
			IF ((VAR_Open = 0.0) AND (NOT VAR_DIFeedBackClose) OR (VAR_Open = 100.0) AND (VAR_DIFeedBackClose)) THEN
				VAR_FaultSensorOff := TRUE;
			ELSE
				VAR_FaultSensorOff := FALSE;
			END_IF
		ELSE
			VAR_FaultSensorOff := FALSE;
		END_IF

		IF IN_ConfigPositionAnalogFBK THEN
			IF (HMI.FBK > HMI.OUT_CV + (HMI.OUT_CV / 10.0) + 5.0) OR (MAX(HMI.FBK, 5.0) < HMI.OUT_CV - (HMI.OUT_CV / 10.0)) THEN
				VAR_FaultSensorFBK := TRUE;
			ELSE
				VAR_FaultSensorFBK := FALSE;
			END_IF
		ELSE
			VAR_FaultSensorFBK := FALSE;
		END_IF

		TMR_TON_PositionFiltered(	IN := VAR_FaultSensorOn OR VAR_FaultSensorOff OR VAR_FaultSensorFBK,
		PT	:= IN_StrokeTime);

		IF (TMR_TON_PositionFiltered.Q OR OUT_FBKFault) AND NOT VAR_Mask THEN
			OUT_Alarm := TRUE;
		ELSIF IN_Reset THEN
			OUT_Alarm := FALSE;
		END_IF

		(*****************************************************************)
		(*****************************RAMP********************************)
		(*****************************************************************)
		IF IN_OpeningRampEn THEN
			VAR_OpeningRamp := IN_OpeningRampValue;
		ELSE
			VAR_OpeningRamp := 100.0;
		END_IF

		IF IN_ClosingRampEn THEN
			VAR_ClosingRamp := IN_ClosingRampValue;
		ELSE
			VAR_ClosingRamp := 100.0;
		END_IF

		LCRMovingRamp(
		enable	:= TRUE,
		x		:= LIMIT(IN_OutMin, VAR_iOpen, IN_OutMax),
		dy_up	:= MAX(0.1, VAR_OpeningRamp),
		dy_down	:= MAX(0.1, VAR_ClosingRamp),
		y_max	:= IN_OutMax,
		y_min	:= IN_OutMin,
		y_set	:= LIMIT(IN_OutMin, VAR_iOpen, IN_OutMax),
		set		:= (NOT IN_ClosingRampEn AND NOT IN_OpeningRampEn)
		);

		VAR_Open := LCRMovingRamp.y;
		OUT_RampDone := LCRMovingRamp.x_reached;

		(*****************************************************************)
		(****************************VALUE SCALING************************)
		(*****************************************************************)
		IF IN_ConfigPositionAnalogFBK THEN
			OUT_FBKFault := (IO.AI_Raw < 6000);
		ELSIF IN_Reset THEN
			OUT_FBKFault := FALSE;
		END_IF

		IF IN_ConfigNormallyOpen THEN
			LCRLimScal_AO(
			x	:= VAR_Open,
			x1	:= 0.0,
			y1	:= 32767.0,
			x2	:= 100.0,
			y2	:= 6553.4,
			);

			LCRLimScal_AI(
			x	:= INT_TO_REAL(IO.AI_Raw),
			x1	:= 32767.0,
			y1	:= 0.0,
			x2	:= 6553.4,
			y2	:= 100.0
			);
		ELSE
			LCRLimScal_AO(
			x	:= VAR_Open,
			x1	:= 0.0,
			y1	:= 6553.4,
			x2	:= 100.0,
			y2	:= 32767.0
			);

			LCRLimScal_AI(
			x	:= INT_TO_REAL(IO.AI_Raw),
			x1	:= 6553.4,
			y1	:= 0.0,
			x2	:= 32767.0,
			y2	:= 100.0
			);
		END_IF
		OUT_Cv		:= VAR_Open;
	ELSE
		OUT_Alarm		:= FALSE;
		OUT_RampDone	:= FALSE;
		OUT_Cv			:= 0.0;
	END_IF

	TMR_TOF_DOValveOn(	IN := VAR_Open > 0.0,
	PT := t#5s);

	VAR_DOValveOn 	:= TMR_TOF_DOValveOn.Q;
	VAR_DOValveOff 	:= NOT VAR_DOValveOn;

	IF IN_ConfigPositionAnalogFBK THEN
		OUT_FBK	:= LCRLimScal_AI.y;
		HMI.FBK := REAL_TO_INT(LCRLimScal_AI.y);
	ELSE
		HMI.FBK := HMI.OUT_CV;
	END_IF
	(*****************************************************************)
	(****************************IO / HMI*****************************)
	(*****************************************************************)
	IO.AO_Raw := REAL_TO_INT(LCRLimScal_AO.y);

	IF NOT IN_Simulation THEN
		IF IN_ConfigNormallyOpen THEN
			IO.Valve.DO_Opened	:= IN_Enable;
			IO.Valve.DO_Closed	:= FALSE;
		ELSE
			IO.Valve.DO_Opened	:= VAR_DOValveOn;
			IO.Valve.DO_Closed	:= VAR_DOValveOff;
		END_IF
	ELSE
		IO.Valve.DO_Opened 	:= FALSE;
		IO.Valve.DO_Closed 	:= FALSE;
		IO.AO_Raw	:= 0;
		IO.AI_Raw	:= REAL_TO_INT(LCRLimScal_AO.y);
	END_IF

	HMI.ManEnable 		:= IN_ManEn;
	HMI.ConfigPresent 	:= IN_ConfigPresent;
	HMI.ConfigPosition 	:= VAR_ConfigPosition;
	HMI.MaskEnable		:= IN_MaskEn;
	HMI.Alarm  			:= OUT_Alarm;
	HMI.Opened 			:= VAR_DOValveOn;
	HMI.Closed 			:= VAR_DOValveOff;
	HMI.Out 			:= VAR_DOValveOn;
	HMI.OUT_CV			:= OUT_Cv;
END_FUNCTION_BLOCK

(* ---- Constant.var ---- *)
VAR CONSTANT
	CST_Valve_Dig_Mono_CFG : USINT := 0;
	CST_Valve_Dig_Bi_CFG : USINT := 1;
	CST_AI_Compare_OFF : USINT := 0; (*FALSE*)
	CST_AI_Compare_LT : USINT := 1; (*PV < SP*)
	CST_AI_Compare_GT : USINT := 2; (*PV > SP*)
	CST_AI_Compare_EQ : USINT := 3; (*PV = SP*)
	CST_AI_Compare_ON : USINT := 4; (*TRUE*)
	CST_AI_FaultMode_Hold : USINT := 0; (*Hold on fault*)
	CST_AI_FaultMode_Low : USINT := 1; (*Low on fault*)
	CST_AI_FaultMode_High : USINT := 2; (*High on fault*)
END_VAR
(*Communication Type*)
VAR CONSTANT
	CST_CFG_NotPresent : USINT := 0;
	CST_CFG_TCP : USINT := 1; (*TCP IP*)
	CST_CFG_ETH : USINT := 2; (*ETHERNET IP*)
	CST_CFG_MODBUS : USINT := 3;
	CST_CFG_PROFIBUS : USINT := 4;
	CST_CFG_POWERLINK : USINT := 5;
	CST_CFG_HW : USINT := 6;
	CST_CFG_UDP : USINT := 7;
	CST_CFG_SCC : USINT := 8;
	CST_CFG_PROFINET : USINT := 9;
	CST_CFG_OPC : USINT := 10;
END_VAR
(*Comparison Constants*)
VAR CONSTANT
	CST_EQ : USINT := 0; (*The equality operator symbol '=' *)
	CST_GE : USINT := 1; (*The greater than or equal to symbol '>=' *)
	CST_LE : USINT := 2; (*The less than or equal to symbol '<='*)
	CST_GT : USINT := 3; (*The greater than operator symbol '>'*)
	CST_LT : USINT := 4; (*The division operator symbol '<'*)
	CST_NE : USINT := 5; (*The unequality operator symbol '<>'*)
END_VAR
